LIN {X 0,Y 586.714,Z 168.831,A -85,B 0,C 180,E1 28018.701,E2 28018.701} C_VEL
LIN {X 0,Y 586.122,Z 408.457,A -85,B 0,C 180,E1 28015.501,E2 28015.501} C_VEL
LIN {X 0,Y 586.025,Z 431.656,A -85,B 0,C 180,E1 28015.125,E2 28015.125} C_VEL
LIN {X 0,Y 585.851,Z 452.374,A -85,B 0,C 180,E1 28014.603,E2 28014.603} C_VEL
LIN {X 0,Y 585.663,Z 472.135,A -85,B 0,C 180,E1 28013.921,E2 28013.921} C_VEL
LIN {X 0,Y 585.449,Z 491.199,A -85,B 0,C 180,E1 28013.077,E2 28013.077} C_VEL
LIN {X 0,Y 585.208,Z 509.397,A -85,B 0,C 180,E1 28012.079,E2 28012.079} C_VEL
LIN {X 0,Y 584.95,Z 527.579,A -85,B 0,C 180,E1 28010.883,E2 28010.883} C_VEL
LIN {X 0,Y 584.711,Z 544.758,A -85,B 0,C 180,E1 28009.536,E2 28009.536} C_VEL
LIN {X 0,Y 584.501,Z 560.932,A -85,B 0,C 180,E1 28008.037,E2 28008.037} C_VEL
LIN {X 0,Y 584.329,Z 575.047,A -85,B 0,C 180,E1 28006.502,E2 28006.502} C_VEL
LIN {X 0,Y 584.202,Z 587.854,A -85,B 0,C 180,E1 28004.876,E2 28004.876} C_VEL
LIN {X 0,Y 584.091,Z 599.923,A -85,B 0,C 180,E1 28003.06,E2 28003.06} C_VEL
LIN {X 0,Y 584.011,Z 610.394,A -85,B 0,C 180,E1 28001.155,E2 28001.155} C_VEL
LIN {X 0,Y 583.958,Z 618.872,A -85,B 0,C 180,E1 27999.262,E2 27999.262} C_VEL
LIN {X 0,Y 583.926,Z 625.897,A -85,B 0,C 180,E1 27997.28,E2 27997.28} C_VEL
LIN {X 0,Y 583.911,Z 631.143,A -85,B 0,C 180,E1 27995.306,E2 27995.306} C_VEL
LIN {X 0,Y 583.905,Z 634.713,A -85,B 0,C 180,E1 27993.336,E2 27993.336} C_VEL
LIN {X 0,Y 583.904,Z 636.639,A -85,B 0,C 180,E1 27991.276,E2 27991.276} C_VEL
LIN {X 0,Y 583.904,Z 636.852,A -85,B 0,C 180,E1 27989.314,E2 27989.314} C_VEL
LIN {X 0,Y 583.91,Z 635.393,A -85,B 0,C 180,E1 27987.253,E2 27987.253} C_VEL
LIN {X 0,Y 583.919,Z 632.17,A -85,B 0,C 180,E1 27985.188,E2 27985.188} C_VEL
LIN {X 0,Y 583.932,Z 627.416,A -85,B 0,C 180,E1 27983.215,E2 27983.215} C_VEL
LIN {X 0,Y 583.952,Z 620.853,A -85,B 0,C 180,E1 27981.235,E2 27981.235} C_VEL
LIN {X 0,Y 583.985,Z 612.797,A -85,B 0,C 180,E1 27979.345,E2 27979.345} C_VEL
LIN {X 0,Y 584.047,Z 602.84,A -85,B 0,C 180,E1 27977.443,E2 27977.443} C_VEL
LIN {X 0,Y 584.154,Z 591.394,A -85,B 0,C 180,E1 27975.63,E2 27975.63} C_VEL
LIN {X 0,Y 584.3,Z 578.453,A -85,B 0,C 180,E1 27973.907,E2 27973.907} C_VEL
LIN {X 0,Y 584.47,Z 563.98,A -85,B 0,C 180,E1 27972.272,E2 27972.272} C_VEL
LIN {X 0,Y 584.684,Z 548.453,A -85,B 0,C 180,E1 27970.781,E2 27970.781} C_VEL
LIN {X 0,Y 584.922,Z 531.283,A -85,B 0,C 180,E1 27969.383,E2 27969.383} C_VEL
LIN {X 0,Y 585.172,Z 512.918,A -85,B 0,C 180,E1 27968.132,E2 27968.132} C_VEL
LIN {X 0,Y 585.387,Z 494.302,A -85,B 0,C 180,E1 27967.082,E2 27967.082} C_VEL
LIN {X 0,Y 585.614,Z 475.711,A -85,B 0,C 180,E1 27966.227,E2 27966.227} C_VEL
LIN {X 0,Y 585.837,Z 455.081,A -85,B 0,C 180,E1 27965.48,E2 27965.48} C_VEL
LIN {X 0,Y 586.013,Z 435.161,A -85,B 0,C 180,E1 27964.947,E2 27964.947} C_VEL
LIN {X 0,Y 586.11,Z 414.501,A -85,B 0,C 180,E1 27964.579,E2 27964.579} C_VEL
LIN {X 0,Y 586.685,Z 176.57,A -85,B 0,C 180,E1 27961.403,E2 27961.403} C_VEL
LIN {X 0,Y 586.477,Z 165.201,A -85,B 0,C 180,E1 27961.237,E2 27961.237} C_VEL
LIN {X 0,Y 586.085,Z 162.496,A -85,B 0,C 180,E1 27961.161,E2 27961.161} C_VEL
LIN {X 0,Y 586.484,Z 115.163,A -85,B 0,C 180,E1 27958.212,E2 27958.212} C_VEL
LIN {X 0,Y 586.557,Z 103.347,A -85,B 0,C 180,E1 27957.46,E2 27957.46} C_VEL
LIN {X 0,Y 584.042,Z 96.734,A -85,B 0,C 180,E1 27956.871,E2 27956.871} C_VEL
LIN {X 0,Y 584.072,Z 96.733,A -85,B 0,C 180,E1 27953.68,E2 27953.68} C_VEL
LIN {X 0,Y 584.05,Z 96.728,A -85,B 0,C 180,E1 27950.696,E2 27950.696} C_VEL
LIN {X 0,Y 584.045,Z 96.731,A -85,B 0,C 180,E1 27947.403,E2 27947.403} C_VEL
LIN {X 0,Y 584.093,Z 96.728,A -85,B 0,C 180,E1 27944.3,E2 27944.3} C_VEL
LIN {X 0,Y 584.035,Z 96.729,A -85,B 0,C 180,E1 27941.127,E2 27941.127} C_VEL
LIN {X 0,Y 584.095,Z 96.723,A -85,B 0,C 180,E1 27938.043,E2 27938.043} C_VEL
LIN {X 0,Y 584.039,Z 96.729,A -85,B 0,C 180,E1 27934.913,E2 27934.913} C_VEL
LIN {X 0,Y 584.045,Z 96.731,A -85,B 0,C 180,E1 27931.591,E2 27931.591} C_VEL
LIN {X 0,Y 584.075,Z 96.727,A -85,B 0,C 180,E1 27928.529,E2 27928.529} C_VEL
LIN {X 0,Y 584.032,Z 96.729,A -85,B 0,C 180,E1 27925.322,E2 27925.322} C_VEL
LIN {X 0,Y 584.096,Z 96.731,A -85,B 0,C 180,E1 27922.17,E2 27922.17} C_VEL
LIN {X 0,Y 584.034,Z 96.727,A -85,B 0,C 180,E1 27919.086,E2 27919.086} C_VEL
LIN {X 0,Y 584.048,Z 96.731,A -85,B 0,C 180,E1 27915.795,E2 27915.795} C_VEL
LIN {X 0,Y 584.048,Z 96.726,A -85,B 0,C 180,E1 27912.859,E2 27912.859} C_VEL
LIN {X 0,Y 584.031,Z 96.73,A -85,B 0,C 180,E1 27909.567,E2 27909.567} C_VEL
LIN {X 0,Y 584.096,Z 96.726,A -85,B 0,C 180,E1 27906.487,E2 27906.487} C_VEL
LIN {X 0,Y 584.027,Z 96.73,A -85,B 0,C 180,E1 27903.337,E2 27903.337} C_VEL
LIN {X 0,Y 584.076,Z 96.731,A -85,B 0,C 180,E1 27900.196,E2 27900.196} C_VEL
LIN {X 0,Y 584.032,Z 96.73,A -85,B 0,C 180,E1 27897.154,E2 27897.154} C_VEL
LIN {X 0,Y 584.032,Z 96.73,A -85,B 0,C 180,E1 27893.808,E2 27893.808} C_VEL
LIN {X 0,Y 584.06,Z 96.73,A -85,B 0,C 180,E1 27890.839,E2 27890.839} C_VEL
LIN {X 0,Y 584.023,Z 96.729,A -85,B 0,C 180,E1 27887.643,E2 27887.643} C_VEL
LIN {X 0,Y 584.077,Z 96.728,A -85,B 0,C 180,E1 27886.731,E2 27886.731} C_VEL
LIN {X 0,Y 583.129,Z 96.853,A -85,B 0,C 180,E1 27885.975,E2 27885.975} C_VEL
LIN {X 0,Y 576.616,Z 97.654,A -85,B 0,C 180,E1 27883.855,E2 27883.855} C_VEL
LIN {X 0,Y 576.087,Z 97.718,A -85,B 0,C 180,E1 27883.302,E2 27883.302} C_VEL
LIN {X 0,Y 576.097,Z 97.721,A -85,B 0,C 180,E1 27880.007,E2 27880.007} C_VEL
LIN {X 0,Y 576.11,Z 97.718,A -85,B 0,C 180,E1 27877.014,E2 27877.014} C_VEL
LIN {X 0,Y 576.084,Z 97.72,A -85,B 0,C 180,E1 27873.805,E2 27873.805} C_VEL
LIN {X 0,Y 576.149,Z 97.717,A -85,B 0,C 180,E1 27870.699,E2 27870.699} C_VEL
LIN {X 0,Y 576.078,Z 97.719,A -85,B 0,C 180,E1 27867.567,E2 27867.567} C_VEL
LIN {X 0,Y 576.128,Z 97.72,A -85,B 0,C 180,E1 27864.452,E2 27864.452} C_VEL
LIN {X 0,Y 576.089,Z 97.72,A -85,B 0,C 180,E1 27861.331,E2 27861.331} C_VEL
LIN {X 0,Y 576.086,Z 97.721,A -85,B 0,C 180,E1 27858.071,E2 27858.071} C_VEL
LIN {X 0,Y 576.115,Z 97.719,A -85,B 0,C 180,E1 27855.06,E2 27855.06} C_VEL
LIN {X 0,Y 576.077,Z 97.722,A -85,B 0,C 180,E1 27851.876,E2 27851.876} C_VEL
LIN {X 0,Y 576.157,Z 97.721,A -85,B 0,C 180,E1 27848.79,E2 27848.79} C_VEL
LIN {X 0,Y 576.08,Z 97.721,A -85,B 0,C 180,E1 27845.673,E2 27845.673} C_VEL
LIN {X 0,Y 576.109,Z 97.724,A -85,B 0,C 180,E1 27842.43,E2 27842.43} C_VEL
LIN {X 0,Y 576.088,Z 97.795,A -85,B 0,C 180,E1 27839.824,E2 27839.824} C_VEL
LIN {X 0,Y 578.546,Z 105.77,A -85,B 0,C 180,E1 27839.016,E2 27839.016} C_VEL
LIN {X 0,Y 577.999,Z 143.994,A -85,B 0,C 180,E1 27835.953,E2 27835.953} C_VEL
LIN {X 0,Y 577.653,Z 175.774,A -85,B 0,C 180,E1 27833.508,E2 27833.508} C_VEL
LIN {X 0,Y 578.35,Z 181.85,A -85,B 0,C 180,E1 27833.398,E2 27833.398} C_VEL
LIN {X 0,Y 577.837,Z 384.429,A -85,B 0,C 180,E1 27830.729,E2 27830.729} C_VEL
LIN {X 0,Y 577.687,Z 403.356,A -85,B 0,C 180,E1 27830.29,E2 27830.29} C_VEL
LIN {X 0,Y 577.5,Z 421.605,A -85,B 0,C 180,E1 27829.678,E2 27829.678} C_VEL
LIN {X 0,Y 577.269,Z 439.198,A -85,B 0,C 180,E1 27828.898,E2 27828.898} C_VEL
LIN {X 0,Y 577.04,Z 455.969,A -85,B 0,C 180,E1 27827.959,E2 27827.959} C_VEL
LIN {X 0,Y 576.809,Z 471.559,A -85,B 0,C 180,E1 27826.891,E2 27826.891} C_VEL
LIN {X 0,Y 576.58,Z 486.636,A -85,B 0,C 180,E1 27825.643,E2 27825.643} C_VEL
LIN {X 0,Y 576.378,Z 500.546,A -85,B 0,C 180,E1 27824.26,E2 27824.26} C_VEL
LIN {X 0,Y 576.212,Z 513.352,A -85,B 0,C 180,E1 27822.73,E2 27822.73} C_VEL
LIN {X 0,Y 576.088,Z 524.59,A -85,B 0,C 180,E1 27821.107,E2 27821.107} C_VEL
LIN {X 0,Y 576.002,Z 534.283,A -85,B 0,C 180,E1 27819.39,E2 27819.39} C_VEL
LIN {X 0,Y 575.957,Z 542,A -85,B 0,C 180,E1 27817.681,E2 27817.681} C_VEL
LIN {X 0,Y 575.927,Z 548.347,A -85,B 0,C 180,E1 27815.856,E2 27815.856} C_VEL
LIN {X 0,Y 575.92,Z 552.989,A -85,B 0,C 180,E1 27813.981,E2 27813.981} C_VEL
LIN {X 0,Y 575.917,Z 555.852,A -85,B 0,C 180,E1 27812.089,E2 27812.089} C_VEL
LIN {X 0,Y 575.911,Z 556.952,A -85,B 0,C 180,E1 27810.198,E2 27810.198} C_VEL
LIN {X 0,Y 575.914,Z 556.311,A -85,B 0,C 180,E1 27808.308,E2 27808.308} C_VEL
LIN {X 0,Y 575.909,Z 553.916,A -85,B 0,C 180,E1 27806.416,E2 27806.416} C_VEL
LIN {X 0,Y 575.922,Z 549.956,A -85,B 0,C 180,E1 27804.62,E2 27804.62} C_VEL
LIN {X 0,Y 575.939,Z 544.27,A -85,B 0,C 180,E1 27802.819,E2 27802.819} C_VEL
LIN {X 0,Y 575.981,Z 537.168,A -85,B 0,C 180,E1 27801.112,E2 27801.112} C_VEL
LIN {X 0,Y 576.056,Z 528.191,A -85,B 0,C 180,E1 27799.398,E2 27799.398} C_VEL
LIN {X 0,Y 576.167,Z 517.752,A -85,B 0,C 180,E1 27797.777,E2 27797.777} C_VEL
LIN {X 0,Y 576.31,Z 505.869,A -85,B 0,C 180,E1 27796.249,E2 27796.249} C_VEL
LIN {X 0,Y 576.498,Z 492.507,A -85,B 0,C 180,E1 27794.817,E2 27794.817} C_VEL
LIN {X 0,Y 576.723,Z 477.51,A -85,B 0,C 180,E1 27793.481,E2 27793.481} C_VEL
LIN {X 0,Y 576.961,Z 461.313,A -85,B 0,C 180,E1 27792.293,E2 27792.293} C_VEL
LIN {X 0,Y 577.198,Z 444.899,A -85,B 0,C 180,E1 27791.308,E2 27791.308} C_VEL
LIN {X 0,Y 577.43,Z 427.61,A -85,B 0,C 180,E1 27790.476,E2 27790.476} C_VEL
LIN {X 0,Y 577.635,Z 409.432,A -85,B 0,C 180,E1 27789.803,E2 27789.803} C_VEL
LIN {X 0,Y 577.794,Z 390.88,A -85,B 0,C 180,E1 27789.311,E2 27789.311} C_VEL
LIN {X 0,Y 577.893,Z 370.714,A -85,B 0,C 180,E1 27788.977,E2 27788.977} C_VEL
LIN {X 0,Y 578.232,Z 179.106,A -85,B 0,C 180,E1 27786.471,E2 27786.471} C_VEL
LIN {X 0,Y 577.601,Z 175.101,A -85,B 0,C 180,E1 27786.375,E2 27786.375} C_VEL
LIN {X 0,Y 578.093,Z 134.758,A -85,B 0,C 180,E1 27783.22,E2 27783.22} C_VEL
LIN {X 0,Y 578.526,Z 105.079,A -85,B 0,C 180,E1 27780.831,E2 27780.831} C_VEL
LIN {X 0,Y 576.084,Z 97.726,A -85,B 0,C 180,E1 27780.066,E2 27780.066} C_VEL
LIN {X 0,Y 576.121,Z 97.719,A -85,B 0,C 180,E1 27776.86,E2 27776.86} C_VEL
LIN {X 0,Y 576.135,Z 97.721,A -85,B 0,C 180,E1 27773.715,E2 27773.715} C_VEL
LIN {X 0,Y 576.115,Z 97.71,A -85,B 0,C 180,E1 27770.562,E2 27770.562} C_VEL
LIN {X 0,Y 576.158,Z 97.714,A -85,B 0,C 180,E1 27767.376,E2 27767.376} C_VEL
LIN {X 0,Y 576.155,Z 97.72,A -85,B 0,C 180,E1 27764.072,E2 27764.072} C_VEL
LIN {X 0,Y 576.14,Z 97.716,A -85,B 0,C 180,E1 27760.733,E2 27760.733} C_VEL
LIN {X 0,Y 576.149,Z 97.713,A -85,B 0,C 180,E1 27757.525,E2 27757.525} C_VEL
LIN {X 0,Y 576.142,Z 97.72,A -85,B 0,C 180,E1 27754.214,E2 27754.214} C_VEL
LIN {X 0,Y 576.158,Z 97.72,A -85,B 0,C 180,E1 27750.909,E2 27750.909} C_VEL
LIN {X 0,Y 576.141,Z 97.757,A -85,B 0,C 180,E1 27749.631,E2 27749.631} C_VEL
LIN {X 0,Y 578.217,Z 105.123,A -85,B 0,C 180,E1 27748.957,E2 27748.957} C_VEL
LIN {X 0,Y 577.914,Z 144.603,A -85,B 0,C 180,E1 27745.886,E2 27745.886} C_VEL
LIN {X 0,Y 577.621,Z 175.862,A -85,B 0,C 180,E1 27743.509,E2 27743.509} C_VEL
LIN {X 0,Y 578.323,Z 181.943,A -85,B 0,C 180,E1 27743.398,E2 27743.398} C_VEL
LIN {X 0,Y 577.84,Z 384.232,A -85,B 0,C 180,E1 27740.732,E2 27740.732} C_VEL
LIN {X 0,Y 577.685,Z 402.976,A -85,B 0,C 180,E1 27740.297,E2 27740.297} C_VEL
LIN {X 0,Y 577.519,Z 420.285,A -85,B 0,C 180,E1 27739.731,E2 27739.731} C_VEL
LIN {X 0,Y 577.286,Z 437.662,A -85,B 0,C 180,E1 27738.972,E2 27738.972} C_VEL
LIN {X 0,Y 577.052,Z 455.018,A -85,B 0,C 180,E1 27738.017,E2 27738.017} C_VEL
LIN {X 0,Y 576.823,Z 471.07,A -85,B 0,C 180,E1 27736.931,E2 27736.931} C_VEL
LIN {X 0,Y 576.585,Z 486.027,A -85,B 0,C 180,E1 27735.695,E2 27735.695} C_VEL
LIN {X 0,Y 576.401,Z 499.639,A -85,B 0,C 180,E1 27734.363,E2 27734.363} C_VEL
LIN {X 0,Y 576.222,Z 512.539,A -85,B 0,C 180,E1 27732.833,E2 27732.833} C_VEL
LIN {X 0,Y 576.102,Z 523.356,A -85,B 0,C 180,E1 27731.306,E2 27731.306} C_VEL
LIN {X 0,Y 576.014,Z 533.232,A -85,B 0,C 180,E1 27729.593,E2 27729.593} C_VEL
LIN {X 0,Y 575.954,Z 541.206,A -85,B 0,C 180,E1 27727.883,E2 27727.883} C_VEL
LIN {X 0,Y 575.927,Z 547.971,A -85,B 0,C 180,E1 27725.979,E2 27725.979} C_VEL
LIN {X 0,Y 575.914,Z 552.591,A -85,B 0,C 180,E1 27724.182,E2 27724.182} C_VEL
LIN {X 0,Y 575.913,Z 555.743,A -85,B 0,C 180,E1 27722.189,E2 27722.189} C_VEL
LIN {X 0,Y 575.913,Z 556.936,A -85,B 0,C 180,E1 27720.299,E2 27720.299} C_VEL
LIN {X 0,Y 575.91,Z 556.313,A -85,B 0,C 180,E1 27718.309,E2 27718.309} C_VEL
LIN {X 0,Y 575.918,Z 554.069,A -85,B 0,C 180,E1 27716.517,E2 27716.517} C_VEL
LIN {X 0,Y 575.922,Z 549.975,A -85,B 0,C 180,E1 27714.621,E2 27714.621} C_VEL
LIN {X 0,Y 575.942,Z 544.257,A -85,B 0,C 180,E1 27712.82,E2 27712.82} C_VEL
LIN {X 0,Y 575.988,Z 536.728,A -85,B 0,C 180,E1 27711.012,E2 27711.012} C_VEL
LIN {X 0,Y 576.058,Z 528.17,A -85,B 0,C 180,E1 27709.398,E2 27709.398} C_VEL
LIN {X 0,Y 576.178,Z 517.139,A -85,B 0,C 180,E1 27707.687,E2 27707.687} C_VEL
LIN {X 0,Y 576.321,Z 504.976,A -85,B 0,C 180,E1 27706.148,E2 27706.148} C_VEL
LIN {X 0,Y 576.511,Z 491.443,A -85,B 0,C 180,E1 27704.715,E2 27704.715} C_VEL
LIN {X 0,Y 576.709,Z 477.443,A -85,B 0,C 180,E1 27703.481,E2 27703.481} C_VEL
LIN {X 0,Y 576.952,Z 462.1,A -85,B 0,C 180,E1 27702.346,E2 27702.346} C_VEL
LIN {X 0,Y 577.177,Z 445.959,A -85,B 0,C 180,E1 27701.368,E2 27701.368} C_VEL
LIN {X 0,Y 577.41,Z 428.793,A -85,B 0,C 180,E1 27700.529,E2 27700.529} C_VEL
LIN {X 0,Y 577.605,Z 411.69,A -85,B 0,C 180,E1 27699.877,E2 27699.877} C_VEL
LIN {X 0,Y 577.766,Z 392.811,A -85,B 0,C 180,E1 27699.355,E2 27699.355} C_VEL
LIN {X 0,Y 577.89,Z 373.954,A -85,B 0,C 180,E1 27699.019,E2 27699.019} C_VEL
LIN {X 0,Y 578.245,Z 179.115,A -85,B 0,C 180,E1 27696.472,E2 27696.472} C_VEL
LIN {X 0,Y 577.585,Z 175.11,A -85,B 0,C 180,E1 27696.375,E2 27696.375} C_VEL
LIN {X 0,Y 577.951,Z 136.16,A -85,B 0,C 180,E1 27693.38,E2 27693.38} C_VEL
LIN {X 0,Y 578.003,Z 114.036,A -85,B 0,C 180,E1 27691.703,E2 27691.703} C_VEL
LIN {X 0,Y 577.718,Z 103.475,A -85,B 0,C 180,E1 27690.928,E2 27690.928} C_VEL
LIN {X 0,Y 576.121,Z 97.721,A -85,B 0,C 180,E1 27690.441,E2 27690.441} C_VEL
LIN {X 0,Y 576.162,Z 97.72,A -85,B 0,C 180,E1 27687.219,E2 27687.219} C_VEL
LIN {X 0,Y 576.133,Z 97.717,A -85,B 0,C 180,E1 27683.962,E2 27683.962} C_VEL
LIN {X 0,Y 576.101,Z 97.72,A -85,B 0,C 180,E1 27680.693,E2 27680.693} C_VEL
LIN {X 0,Y 576.153,Z 97.721,A -85,B 0,C 180,E1 27677.523,E2 27677.523} C_VEL
LIN {X 0,Y 576.094,Z 97.721,A -85,B 0,C 180,E1 27674.383,E2 27674.383} C_VEL
LIN {X 0,Y 576.084,Z 97.722,A -85,B 0,C 180,E1 27671.001,E2 27671.001} C_VEL
LIN {X 0,Y 576.153,Z 97.721,A -85,B 0,C 180,E1 27667.904,E2 27667.904} C_VEL
LIN {X 0,Y 576.096,Z 97.723,A -85,B 0,C 180,E1 27664.7,E2 27664.7} C_VEL
LIN {X 0,Y 576.135,Z 97.75,A -85,B 0,C 180,E1 27663.573,E2 27663.573} C_VEL
LIN {X 0,Y 579.556,Z 106.935,A -85,B 0,C 180,E1 27662.748,E2 27662.748} C_VEL
LIN {X 0,Y 578.949,Z 154.809,A -85,B 0,C 180,E1 27659.714,E2 27659.714} C_VEL
LIN {X 0,Y 578.961,Z 163.557,A -85,B 0,C 180,E1 27659.195,E2 27659.195} C_VEL
LIN {X 0,Y 579.691,Z 169.722,A -85,B 0,C 180,E1 27659.069,E2 27659.069} C_VEL
LIN {X 0,Y 578.899,Z 409.209,A -85,B 0,C 180,E1 27655.832,E2 27655.832} C_VEL
LIN {X 0,Y 578.766,Z 431.846,A -85,B 0,C 180,E1 27655.459,E2 27655.459} C_VEL
LIN {X 0,Y 578.532,Z 452.639,A -85,B 0,C 180,E1 27654.927,E2 27654.927} C_VEL
LIN {X 0,Y 578.29,Z 472.133,A -85,B 0,C 180,E1 27654.245,E2 27654.245} C_VEL
LIN {X 0,Y 577.996,Z 491.203,A -85,B 0,C 180,E1 27653.392,E2 27653.392} C_VEL
LIN {X 0,Y 577.66,Z 510.29,A -85,B 0,C 180,E1 27652.33,E2 27652.33} C_VEL
LIN {X 0,Y 577.326,Z 527.635,A -85,B 0,C 180,E1 27651.168,E2 27651.168} C_VEL
LIN {X 0,Y 577.008,Z 544.936,A -85,B 0,C 180,E1 27649.792,E2 27649.792} C_VEL
LIN {X 0,Y 576.715,Z 561.438,A -85,B 0,C 180,E1 27648.237,E2 27648.237} C_VEL
LIN {X 0,Y 576.472,Z 575.897,A -85,B 0,C 180,E1 27646.63,E2 27646.63} C_VEL
LIN {X 0,Y 576.284,Z 589.161,A -85,B 0,C 180,E1 27644.895,E2 27644.895} C_VEL
LIN {X 0,Y 576.149,Z 600.524,A -85,B 0,C 180,E1 27643.141,E2 27643.141} C_VEL
LIN {X 0,Y 576.043,Z 610.908,A -85,B 0,C 180,E1 27641.21,E2 27641.21} C_VEL
LIN {X 0,Y 575.973,Z 619.278,A -85,B 0,C 180,E1 27639.291,E2 27639.291} C_VEL
LIN {X 0,Y 575.932,Z 625.897,A -85,B 0,C 180,E1 27637.382,E2 27637.382} C_VEL
LIN {X 0,Y 575.912,Z 631.143,A -85,B 0,C 180,E1 27635.38,E2 27635.38} C_VEL
LIN {X 0,Y 575.906,Z 634.745,A -85,B 0,C 180,E1 27633.357,E2 27633.357} C_VEL
LIN {X 0,Y 575.903,Z 636.639,A -85,B 0,C 180,E1 27631.294,E2 27631.294} C_VEL
LIN {X 0,Y 575.904,Z 636.852,A -85,B 0,C 180,E1 27629.304,E2 27629.304} C_VEL
LIN {X 0,Y 575.912,Z 635.393,A -85,B 0,C 180,E1 27627.214,E2 27627.214} C_VEL
LIN {X 0,Y 575.921,Z 632.17,A -85,B 0,C 180,E1 27625.121,E2 27625.121} C_VEL
LIN {X 0,Y 575.938,Z 627.416,A -85,B 0,C 180,E1 27623.121,E2 27623.121} C_VEL
LIN {X 0,Y 575.967,Z 620.853,A -85,B 0,C 180,E1 27621.113,E2 27621.113} C_VEL
LIN {X 0,Y 576.017,Z 612.797,A -85,B 0,C 180,E1 27619.196,E2 27619.196} C_VEL
LIN {X 0,Y 576.102,Z 602.842,A -85,B 0,C 180,E1 27617.267,E2 27617.267} C_VEL
LIN {X 0,Y 576.247,Z 591.395,A -85,B 0,C 180,E1 27615.429,E2 27615.429} C_VEL
LIN {X 0,Y 576.439,Z 578.452,A -85,B 0,C 180,E1 27613.681,E2 27613.681} C_VEL
LIN {X 0,Y 576.673,Z 563.98,A -85,B 0,C 180,E1 27612.024,E2 27612.024} C_VEL
LIN {X 0,Y 576.961,Z 548.486,A -85,B 0,C 180,E1 27610.516,E2 27610.516} C_VEL
LIN {X 0,Y 577.284,Z 531.284,A -85,B 0,C 180,E1 27609.097,E2 27609.097} C_VEL
LIN {X 0,Y 577.624,Z 512.914,A -85,B 0,C 180,E1 27607.831,E2 27607.831} C_VEL
LIN {X 0,Y 577.925,Z 494.298,A -85,B 0,C 180,E1 27606.769,E2 27606.769} C_VEL
LIN {X 0,Y 578.224,Z 475.18,A -85,B 0,C 180,E1 27605.881,E2 27605.881} C_VEL
LIN {X 0,Y 578.517,Z 454.709,A -85,B 0,C 180,E1 27605.137,E2 27605.137} C_VEL
LIN {X 0,Y 578.752,Z 434.609,A -85,B 0,C 180,E1 27604.599,E2 27604.599} C_VEL
LIN {X 0,Y 578.886,Z 413.866,A -85,B 0,C 180,E1 27604.23,E2 27604.23} C_VEL
LIN {X 0,Y 579.665,Z 175.552,A -85,B 0,C 180,E1 27601.01,E2 27601.01} C_VEL
LIN {X 0,Y 579.444,Z 166.395,A -85,B 0,C 180,E1 27600.871,E2 27600.871} C_VEL
LIN {X 0,Y 578.855,Z 162.496,A -85,B 0,C 180,E1 27600.766,E2 27600.766} C_VEL
LIN {X 0,Y 579.405,Z 116.064,A -85,B 0,C 180,E1 27597.835,E2 27597.835} C_VEL
LIN {X 0,Y 579.556,Z 106.958,A -85,B 0,C 180,E1 27597.253,E2 27597.253} C_VEL
LIN {X 0,Y 576.134,Z 97.72,A -85,B 0,C 180,E1 27596.41,E2 27596.41} C_VEL
LIN {X 0,Y 576.102,Z 97.721,A -85,B 0,C 180,E1 27593.219,E2 27593.219} C_VEL
LIN {X 0,Y 576.164,Z 97.718,A -85,B 0,C 180,E1 27590.053,E2 27590.053} C_VEL
LIN {X 0,Y 576.103,Z 97.719,A -85,B 0,C 180,E1 27586.859,E2 27586.859} C_VEL
LIN {X 0,Y 576.108,Z 97.718,A -85,B 0,C 180,E1 27583.495,E2 27583.495} C_VEL
LIN {X 0,Y 576.152,Z 97.716,A -85,B 0,C 180,E1 27580.339,E2 27580.339} C_VEL
LIN {X 0,Y 576.095,Z 97.715,A -85,B 0,C 180,E1 27577.155,E2 27577.155} C_VEL
LIN {X 0,Y 576.143,Z 97.718,A -85,B 0,C 180,E1 27573.95,E2 27573.95} C_VEL
LIN {X 0,Y 576.102,Z 97.718,A -85,B 0,C 180,E1 27570.912,E2 27570.912} C_VEL
LIN {X 0,Y 576.101,Z 97.719,A -85,B 0,C 180,E1 27567.519,E2 27567.519} C_VEL
LIN {X 0,Y 576.151,Z 97.717,A -85,B 0,C 180,E1 27564.395,E2 27564.395} C_VEL
LIN {X 0,Y 576.092,Z 97.719,A -85,B 0,C 180,E1 27561.252,E2 27561.252} C_VEL
LIN {X 0,Y 576.144,Z 97.72,A -85,B 0,C 180,E1 27558.098,E2 27558.098} C_VEL
LIN {X 0,Y 576.1,Z 97.718,A -85,B 0,C 180,E1 27554.987,E2 27554.987} C_VEL
LIN {X 0,Y 576.095,Z 97.719,A -85,B 0,C 180,E1 27551.614,E2 27551.614} C_VEL
LIN {X 0,Y 576.152,Z 97.718,A -85,B 0,C 180,E1 27548.482,E2 27548.482} C_VEL
LIN {X 0,Y 576.088,Z 97.719,A -85,B 0,C 180,E1 27545.378,E2 27545.378} C_VEL
LIN {X 0,Y 576.137,Z 97.717,A -85,B 0,C 180,E1 27542.188,E2 27542.188} C_VEL
LIN {X 0,Y 576.095,Z 97.718,A -85,B 0,C 180,E1 27539.105,E2 27539.105} C_VEL
LIN {X 0,Y 576.095,Z 97.718,A -85,B 0,C 180,E1 27535.82,E2 27535.82} C_VEL
LIN {X 0,Y 576.122,Z 97.717,A -85,B 0,C 180,E1 27532.822,E2 27532.822} C_VEL
LIN {X 0,Y 576.084,Z 97.718,A -85,B 0,C 180,E1 27529.601,E2 27529.601} C_VEL
LIN {X 0,Y 576.154,Z 97.72,A -85,B 0,C 180,E1 27526.451,E2 27526.451} C_VEL
LIN {X 0,Y 576.087,Z 97.718,A -85,B 0,C 180,E1 27523.302,E2 27523.302} C_VEL
LIN {X 0,Y 575.122,Z 97.845,A -85,B 0,C 180,E1 27522.536,E2 27522.536} C_VEL
LIN {X 0,Y 568.601,Z 98.659,A -85,B 0,C 180,E1 27520.33,E2 27520.33} C_VEL
LIN {X 0,Y 568.148,Z 98.709,A -85,B 0,C 180,E1 27519.825,E2 27519.825} C_VEL
LIN {X 0,Y 568.211,Z 98.705,A -85,B 0,C 180,E1 27516.676,E2 27516.676} C_VEL
LIN {X 0,Y 568.142,Z 98.709,A -85,B 0,C 180,E1 27513.561,E2 27513.561} C_VEL
LIN {X 0,Y 568.185,Z 98.71,A -85,B 0,C 180,E1 27510.364,E2 27510.364} C_VEL
LIN {X 0,Y 568.153,Z 98.708,A -85,B 0,C 180,E1 27507.266,E2 27507.266} C_VEL
LIN {X 0,Y 568.146,Z 98.709,A -85,B 0,C 180,E1 27503.999,E2 27503.999} C_VEL
LIN {X 0,Y 568.204,Z 98.709,A -85,B 0,C 180,E1 27500.822,E2 27500.822} C_VEL
LIN {X 0,Y 568.137,Z 98.71,A -85,B 0,C 180,E1 27497.658,E2 27497.658} C_VEL
LIN {X 0,Y 568.179,Z 98.711,A -85,B 0,C 180,E1 27494.457,E2 27494.457} C_VEL
LIN {X 0,Y 568.148,Z 98.711,A -85,B 0,C 180,E1 27491.429,E2 27491.429} C_VEL
LIN {X 0,Y 568.147,Z 98.709,A -85,B 0,C 180,E1 27488.125,E2 27488.125} C_VEL
LIN {X 0,Y 568.196,Z 98.709,A -85,B 0,C 180,E1 27485.005,E2 27485.005} C_VEL
LIN {X 0,Y 568.14,Z 98.714,A -85,B 0,C 180,E1 27481.867,E2 27481.867} C_VEL
LIN {X 0,Y 568.181,Z 98.929,A -85,B 0,C 180,E1 27480.226,E2 27480.226} C_VEL
LIN {X 0,Y 571.286,Z 108.519,A -85,B 0,C 180,E1 27479.228,E2 27479.228} C_VEL
LIN {X 0,Y 570.598,Z 147.207,A -85,B 0,C 180,E1 27476.092,E2 27476.092} C_VEL
LIN {X 0,Y 570.154,Z 175.718,A -85,B 0,C 180,E1 27473.852,E2 27473.852} C_VEL
LIN {X 0,Y 571.026,Z 182.769,A -85,B 0,C 180,E1 27473.71,E2 27473.71} C_VEL
LIN {X 0,Y 570.356,Z 384.462,A -85,B 0,C 180,E1 27471.014,E2 27471.014} C_VEL
LIN {X 0,Y 570.165,Z 403.441,A -85,B 0,C 180,E1 27470.568,E2 27470.568} C_VEL
LIN {X 0,Y 569.93,Z 421.618,A -85,B 0,C 180,E1 27469.951,E2 27469.951} C_VEL
LIN {X 0,Y 569.64,Z 439.206,A -85,B 0,C 180,E1 27469.161,E2 27469.161} C_VEL
LIN {X 0,Y 569.347,Z 455.902,A -85,B 0,C 180,E1 27468.215,E2 27468.215} C_VEL
LIN {X 0,Y 569.044,Z 472.093,A -85,B 0,C 180,E1 27467.087,E2 27467.087} C_VEL
LIN {X 0,Y 568.754,Z 487.196,A -85,B 0,C 180,E1 27465.812,E2 27465.812} C_VEL
LIN {X 0,Y 568.515,Z 500.551,A -85,B 0,C 180,E1 27464.461,E2 27464.461} C_VEL
LIN {X 0,Y 568.302,Z 513.357,A -85,B 0,C 180,E1 27462.91,E2 27462.91} C_VEL
LIN {X 0,Y 568.138,Z 524.593,A -85,B 0,C 180,E1 27461.264,E2 27461.264} C_VEL
LIN {X 0,Y 568.028,Z 534.286,A -85,B 0,C 180,E1 27459.523,E2 27459.523} C_VEL
LIN {X 0,Y 567.968,Z 542.002,A -85,B 0,C 180,E1 27457.79,E2 27457.79} C_VEL
LIN {X 0,Y 567.933,Z 548.282,A -85,B 0,C 180,E1 27455.961,E2 27455.961} C_VEL
LIN {X 0,Y 567.919,Z 552.787,A -85,B 0,C 180,E1 27454.139,E2 27454.139} C_VEL
LIN {X 0,Y 567.915,Z 555.743,A -85,B 0,C 180,E1 27452.219,E2 27452.219} C_VEL
LIN {X 0,Y 567.909,Z 556.93,A -85,B 0,C 180,E1 27450.302,E2 27450.302} C_VEL
LIN {X 0,Y 567.914,Z 556.378,A -85,B 0,C 180,E1 27448.385,E2 27448.385} C_VEL
LIN {X 0,Y 567.908,Z 554.074,A -85,B 0,C 180,E1 27446.467,E2 27446.467} C_VEL
LIN {X 0,Y 567.924,Z 550.208,A -85,B 0,C 180,E1 27444.645,E2 27444.645} C_VEL
LIN {X 0,Y 567.945,Z 544.62,A -85,B 0,C 180,E1 27442.819,E2 27442.819} C_VEL
LIN {X 0,Y 567.998,Z 537.626,A -85,B 0,C 180,E1 27441.088,E2 27441.088} C_VEL
LIN {X 0,Y 568.091,Z 528.765,A -85,B 0,C 180,E1 27439.35,E2 27439.35} C_VEL
LIN {X 0,Y 568.229,Z 518.454,A -85,B 0,C 180,E1 27437.706,E2 27437.706} C_VEL
LIN {X 0,Y 568.406,Z 506.713,A -85,B 0,C 180,E1 27436.158,E2 27436.158} C_VEL
LIN {X 0,Y 568.639,Z 493.513,A -85,B 0,C 180,E1 27434.707,E2 27434.707} C_VEL
LIN {X 0,Y 568.92,Z 478.736,A -85,B 0,C 180,E1 27433.353,E2 27433.353} C_VEL
LIN {X 0,Y 569.224,Z 462.866,A -85,B 0,C 180,E1 27432.15,E2 27432.15} C_VEL
LIN {X 0,Y 569.536,Z 445.883,A -85,B 0,C 180,E1 27431.1,E2 27431.1} C_VEL
LIN {X 0,Y 569.826,Z 428.863,A -85,B 0,C 180,E1 27430.258,E2 27430.258} C_VEL
LIN {X 0,Y 570.091,Z 410.245,A -85,B 0,C 180,E1 27429.55,E2 27429.55} C_VEL
LIN {X 0,Y 570.295,Z 391.496,A -85,B 0,C 180,E1 27429.04,E2 27429.04} C_VEL
LIN {X 0,Y 570.421,Z 371.554,A -85,B 0,C 180,E1 27428.7,E2 27428.7} C_VEL
LIN {X 0,Y 570.928,Z 180.337,A -85,B 0,C 180,E1 27426.161,E2 27426.161} C_VEL
LIN {X 0,Y 570.09,Z 175.035,A -85,B 0,C 180,E1 27426.031,E2 27426.031} C_VEL
LIN {X 0,Y 570.769,Z 135.339,A -85,B 0,C 180,E1 27422.861,E2 27422.861} C_VEL
LIN {X 0,Y 571.288,Z 108.097,A -85,B 0,C 180,E1 27420.645,E2 27420.645} C_VEL
LIN {X 0,Y 568.169,Z 98.715,A -85,B 0,C 180,E1 27419.635,E2 27419.635} C_VEL
LIN {X 0,Y 568.156,Z 98.709,A -85,B 0,C 180,E1 27416.455,E2 27416.455} C_VEL
LIN {X 0,Y 568.222,Z 98.708,A -85,B 0,C 180,E1 27413.253,E2 27413.253} C_VEL
LIN {X 0,Y 568.197,Z 98.701,A -85,B 0,C 180,E1 27409.949,E2 27409.949} C_VEL
LIN {X 0,Y 568.186,Z 98.704,A -85,B 0,C 180,E1 27406.617,E2 27406.617} C_VEL
LIN {X 0,Y 568.218,Z 98.7,A -85,B 0,C 180,E1 27403.335,E2 27403.335} C_VEL
LIN {X 0,Y 568.213,Z 98.707,A -85,B 0,C 180,E1 27399.962,E2 27399.962} C_VEL
LIN {X 0,Y 568.214,Z 98.707,A -85,B 0,C 180,E1 27396.622,E2 27396.622} C_VEL
LIN {X 0,Y 568.218,Z 98.703,A -85,B 0,C 180,E1 27393.297,E2 27393.297} C_VEL
LIN {X 0,Y 568.185,Z 98.71,A -85,B 0,C 180,E1 27389.985,E2 27389.985} C_VEL
LIN {X 0,Y 570.781,Z 107.539,A -85,B 0,C 180,E1 27389.143,E2 27389.143} C_VEL
LIN {X 0,Y 570.435,Z 146.471,A -85,B 0,C 180,E1 27386.101,E2 27386.101} C_VEL
LIN {X 0,Y 570.08,Z 175.861,A -85,B 0,C 180,E1 27383.837,E2 27383.837} C_VEL
LIN {X 0,Y 570.98,Z 182.871,A -85,B 0,C 180,E1 27383.705,E2 27383.705} C_VEL
LIN {X 0,Y 570.356,Z 384.027,A -85,B 0,C 180,E1 27381.02,E2 27381.02} C_VEL
LIN {X 0,Y 570.167,Z 402.675,A -85,B 0,C 180,E1 27380.586,E2 27380.586} C_VEL
LIN {X 0,Y 569.952,Z 420.3,A -85,B 0,C 180,E1 27380.004,E2 27380.004} C_VEL
LIN {X 0,Y 569.666,Z 437.016,A -85,B 0,C 180,E1 27379.267,E2 27379.267} C_VEL
LIN {X 0,Y 569.378,Z 454.19,A -85,B 0,C 180,E1 27378.321,E2 27378.321} C_VEL
LIN {X 0,Y 569.086,Z 469.632,A -85,B 0,C 180,E1 27377.273,E2 27377.273} C_VEL
LIN {X 0,Y 568.789,Z 484.888,A -85,B 0,C 180,E1 27376.021,E2 27376.021} C_VEL
LIN {X 0,Y 568.547,Z 498.312,A -85,B 0,C 180,E1 27374.705,E2 27374.705} C_VEL
LIN {X 0,Y 568.336,Z 510.984,A -85,B 0,C 180,E1 27373.221,E2 27373.221} C_VEL
LIN {X 0,Y 568.178,Z 521.984,A -85,B 0,C 180,E1 27371.676,E2 27371.676} C_VEL
LIN {X 0,Y 568.054,Z 532.2,A -85,B 0,C 180,E1 27369.933,E2 27369.933} C_VEL
LIN {X 0,Y 567.985,Z 539.918,A -85,B 0,C 180,E1 27368.3,E2 27368.3} C_VEL
LIN {X 0,Y 567.946,Z 546.764,A -85,B 0,C 180,E1 27366.47,E2 27366.47} C_VEL
LIN {X 0,Y 567.919,Z 551.704,A -85,B 0,C 180,E1 27364.645,E2 27364.645} C_VEL
LIN {X 0,Y 567.915,Z 555.026,A -85,B 0,C 180,E1 27362.826,E2 27362.826} C_VEL
LIN {X 0,Y 567.909,Z 556.748,A -85,B 0,C 180,E1 27360.908,E2 27360.908} C_VEL
LIN {X 0,Y 567.912,Z 556.788,A -85,B 0,C 180,E1 27359.092,E2 27359.092} C_VEL
LIN {X 0,Y 567.909,Z 555.143,A -85,B 0,C 180,E1 27357.175,E2 27357.175} C_VEL
LIN {X 0,Y 567.922,Z 551.906,A -85,B 0,C 180,E1 27355.355,E2 27355.355} C_VEL
LIN {X 0,Y 567.942,Z 546.718,A -85,B 0,C 180,E1 27353.429,E2 27353.429} C_VEL
LIN {X 0,Y 567.977,Z 540.296,A -85,B 0,C 180,E1 27351.7,E2 27351.7} C_VEL
LIN {X 0,Y 568.057,Z 532.162,A -85,B 0,C 180,E1 27349.965,E2 27349.965} C_VEL
LIN {X 0,Y 568.171,Z 522.561,A -85,B 0,C 180,E1 27348.324,E2 27348.324} C_VEL
LIN {X 0,Y 568.327,Z 511.695,A -85,B 0,C 180,E1 27346.779,E2 27346.779} C_VEL
LIN {X 0,Y 568.536,Z 499.183,A -85,B 0,C 180,E1 27345.299,E2 27345.299} C_VEL
LIN {X 0,Y 568.774,Z 485.881,A -85,B 0,C 180,E1 27343.979,E2 27343.979} C_VEL
LIN {X 0,Y 569.073,Z 470.112,A -85,B 0,C 180,E1 27342.674,E2 27342.674} C_VEL
LIN {X 0,Y 569.385,Z 453.993,A -85,B 0,C 180,E1 27341.574,E2 27341.574} C_VEL
LIN {X 0,Y 569.669,Z 437.221,A -85,B 0,C 180,E1 27340.653,E2 27340.653} C_VEL
LIN {X 0,Y 569.958,Z 419.848,A -85,B 0,C 180,E1 27339.889,E2 27339.889} C_VEL
LIN {X 0,Y 570.173,Z 401.862,A -85,B 0,C 180,E1 27339.301,E2 27339.301} C_VEL
LIN {X 0,Y 570.362,Z 382.31,A -85,B 0,C 180,E1 27338.863,E2 27338.863} C_VEL
LIN {X 0,Y 570.886,Z 180.226,A -85,B 0,C 180,E1 27336.166,E2 27336.166} C_VEL
LIN {X 0,Y 570.06,Z 175.093,A -85,B 0,C 180,E1 27336.038,E2 27336.038} C_VEL
LIN {X 0,Y 570.413,Z 144.512,A -85,B 0,C 180,E1 27333.674,E2 27333.674} C_VEL
LIN {X 0,Y 570.41,Z 111.791,A -85,B 0,C 180,E1 27331.216,E2 27331.216} C_VEL
LIN {X 0,Y 570.308,Z 106.324,A -85,B 0,C 180,E1 27330.82,E2 27330.82} C_VEL
LIN {X 0,Y 568.186,Z 98.709,A -85,B 0,C 180,E1 27330.176,E2 27330.176} C_VEL
LIN {X 0,Y 568.186,Z 98.71,A -85,B 0,C 180,E1 27326.82,E2 27326.82} C_VEL
LIN {X 0,Y 568.219,Z 98.707,A -85,B 0,C 180,E1 27323.63,E2 27323.63} C_VEL
LIN {X 0,Y 568.164,Z 98.708,A -85,B 0,C 180,E1 27320.426,E2 27320.426} C_VEL
LIN {X 0,Y 568.18,Z 98.711,A -85,B 0,C 180,E1 27317.208,E2 27317.208} C_VEL
LIN {X 0,Y 568.175,Z 98.71,A -85,B 0,C 180,E1 27314.112,E2 27314.112} C_VEL
LIN {X 0,Y 568.142,Z 98.711,A -85,B 0,C 180,E1 27310.895,E2 27310.895} C_VEL
LIN {X 0,Y 568.214,Z 98.71,A -85,B 0,C 180,E1 27307.761,E2 27307.761} C_VEL
LIN {X 0,Y 568.165,Z 98.713,A -85,B 0,C 180,E1 27304.555,E2 27304.555} C_VEL
LIN {X 0,Y 568.24,Z 98.911,A -85,B 0,C 180,E1 27304.025,E2 27304.025} C_VEL
LIN {X 0,Y 572.481,Z 110.542,A -85,B 0,C 180,E1 27302.966,E2 27302.966} C_VEL
LIN {X 0,Y 571.732,Z 157.514,A -85,B 0,C 180,E1 27299.954,E2 27299.954} C_VEL
LIN {X 0,Y 571.759,Z 163.574,A -85,B 0,C 180,E1 27299.599,E2 27299.599} C_VEL
LIN {X 0,Y 572.693,Z 170.74,A -85,B 0,C 180,E1 27299.445,E2 27299.445} C_VEL
LIN {X 0,Y 571.696,Z 409.602,A -85,B 0,C 180,E1 27296.177,E2 27296.177} C_VEL
LIN {X 0,Y 571.527,Z 432.033,A -85,B 0,C 180,E1 27295.801,E2 27295.801} C_VEL
LIN {X 0,Y 571.233,Z 452.995,A -85,B 0,C 180,E1 27295.257,E2 27295.257} C_VEL
LIN {X 0,Y 570.935,Z 472.13,A -85,B 0,C 180,E1 27294.578,E2 27294.578} C_VEL
LIN {X 0,Y 570.562,Z 491.206,A -85,B 0,C 180,E1 27293.715,E2 27293.715} C_VEL
LIN {X 0,Y 570.133,Z 510.294,A -85,B 0,C 180,E1 27292.641,E2 27292.641} C_VEL
LIN {X 0,Y 569.725,Z 527.638,A -85,B 0,C 180,E1 27291.464,E2 27291.464} C_VEL
LIN {X 0,Y 569.326,Z 544.822,A -85,B 0,C 180,E1 27290.081,E2 27290.081} C_VEL
LIN {X 0,Y 568.949,Z 561.438,A -85,B 0,C 180,E1 27288.495,E2 27288.495} C_VEL
LIN {X 0,Y 568.64,Z 575.898,A -85,B 0,C 180,E1 27286.866,E2 27286.866} C_VEL
LIN {X 0,Y 568.408,Z 588.562,A -85,B 0,C 180,E1 27285.195,E2 27285.195} C_VEL
LIN {X 0,Y 568.212,Z 600.526,A -85,B 0,C 180,E1 27283.328,E2 27283.328} C_VEL
LIN {X 0,Y 568.078,Z 610.907,A -85,B 0,C 180,E1 27281.37,E2 27281.37} C_VEL
LIN {X 0,Y 567.989,Z 619.278,A -85,B 0,C 180,E1 27279.423,E2 27279.423} C_VEL
LIN {X 0,Y 567.937,Z 626.2,A -85,B 0,C 180,E1 27277.385,E2 27277.385} C_VEL
LIN {X 0,Y 567.914,Z 631.554,A -85,B 0,C 180,E1 27275.253,E2 27275.253} C_VEL
LIN {X 0,Y 567.908,Z 634.942,A -85,B 0,C 180,E1 27273.23,E2 27273.23} C_VEL
LIN {X 0,Y 567.91,Z 636.759,A -85,B 0,C 180,E1 27271.11,E2 27271.11} C_VEL
LIN {X 0,Y 567.914,Z 636.784,A -85,B 0,C 180,E1 27268.992,E2 27268.992} C_VEL
LIN {X 0,Y 567.914,Z 635.17,A -85,B 0,C 180,E1 27266.973,E2 27266.973} C_VEL
LIN {X 0,Y 567.916,Z 631.761,A -85,B 0,C 180,E1 27264.849,E2 27264.849} C_VEL
LIN {X 0,Y 567.938,Z 626.811,A -85,B 0,C 180,E1 27262.82,E2 27262.82} C_VEL
LIN {X 0,Y 567.987,Z 620.492,A -85,B 0,C 180,E1 27260.885,E2 27260.885} C_VEL
LIN {X 0,Y 568.06,Z 612.337,A -85,B 0,C 180,E1 27258.94,E2 27258.94} C_VEL
LIN {X 0,Y 568.166,Z 602.843,A -85,B 0,C 180,E1 27257.086,E2 27257.086} C_VEL
LIN {X 0,Y 568.349,Z 591.396,A -85,B 0,C 180,E1 27255.222,E2 27255.222} C_VEL
LIN {X 0,Y 568.585,Z 578.451,A -85,B 0,C 180,E1 27253.449,E2 27253.449} C_VEL
LIN {X 0,Y 568.889,Z 563.98,A -85,B 0,C 180,E1 27251.77,E2 27251.77} C_VEL
LIN {X 0,Y 569.247,Z 548.457,A -85,B 0,C 180,E1 27250.239,E2 27250.239} C_VEL
LIN {X 0,Y 569.658,Z 531.285,A -85,B 0,C 180,E1 27248.804,E2 27248.804} C_VEL
LIN {X 0,Y 570.088,Z 512.911,A -85,B 0,C 180,E1 27247.522,E2 27247.522} C_VEL
LIN {X 0,Y 570.486,Z 494.124,A -85,B 0,C 180,E1 27246.438,E2 27246.438} C_VEL
LIN {X 0,Y 570.867,Z 474.728,A -85,B 0,C 180,E1 27245.53,E2 27245.53} C_VEL
LIN {X 0,Y 571.222,Z 454.089,A -85,B 0,C 180,E1 27244.778,E2 27244.778} C_VEL
LIN {X 0,Y 571.518,Z 433.4,A -85,B 0,C 180,E1 27244.228,E2 27244.228} C_VEL
LIN {X 0,Y 571.686,Z 412.34,A -85,B 0,C 180,E1 27243.86,E2 27243.86} C_VEL
LIN {X 0,Y 572.679,Z 173.154,A -85,B 0,C 180,E1 27240.588,E2 27240.588} C_VEL
LIN {X 0,Y 572.404,Z 167.387,A -85,B 0,C 180,E1 27240.491,E2 27240.491} C_VEL
LIN {X 0,Y 571.651,Z 162.729,A -85,B 0,C 180,E1 27240.376,E2 27240.376} C_VEL
LIN {X 0,Y 572.368,Z 116.063,A -85,B 0,C 180,E1 27237.391,E2 27237.391} C_VEL
LIN {X 0,Y 572.356,Z 109.753,A -85,B 0,C 180,E1 27236.974,E2 27236.974} C_VEL
LIN {X 0,Y 568.223,Z 98.708,A -85,B 0,C 180,E1 27235.948,E2 27235.948} C_VEL
LIN {X 0,Y 568.171,Z 98.709,A -85,B 0,C 180,E1 27232.746,E2 27232.746} C_VEL
LIN {X 0,Y 568.166,Z 98.708,A -85,B 0,C 180,E1 27229.33,E2 27229.33} C_VEL
LIN {X 0,Y 568.223,Z 98.707,A -85,B 0,C 180,E1 27226.11,E2 27226.11} C_VEL
LIN {X 0,Y 568.161,Z 98.705,A -85,B 0,C 180,E1 27222.925,E2 27222.925} C_VEL
LIN {X 0,Y 568.171,Z 98.699,A -85,B 0,C 180,E1 27219.571,E2 27219.571} C_VEL
LIN {X 0,Y 568.198,Z 98.701,A -85,B 0,C 180,E1 27216.47,E2 27216.47} C_VEL
LIN {X 0,Y 568.156,Z 98.705,A -85,B 0,C 180,E1 27213.29,E2 27213.29} C_VEL
LIN {X 0,Y 568.218,Z 98.708,A -85,B 0,C 180,E1 27210.099,E2 27210.099} C_VEL
LIN {X 0,Y 568.16,Z 98.707,A -85,B 0,C 180,E1 27207.003,E2 27207.003} C_VEL
LIN {X 0,Y 568.166,Z 98.707,A -85,B 0,C 180,E1 27203.655,E2 27203.655} C_VEL
LIN {X 0,Y 568.195,Z 98.707,A -85,B 0,C 180,E1 27200.585,E2 27200.585} C_VEL
LIN {X 0,Y 568.153,Z 98.707,A -85,B 0,C 180,E1 27197.408,E2 27197.408} C_VEL
LIN {X 0,Y 568.22,Z 98.705,A -85,B 0,C 180,E1 27194.261,E2 27194.261} C_VEL
LIN {X 0,Y 568.152,Z 98.708,A -85,B 0,C 180,E1 27191.162,E2 27191.162} C_VEL
LIN {X 0,Y 568.172,Z 98.704,A -85,B 0,C 180,E1 27187.889,E2 27187.889} C_VEL
LIN {X 0,Y 568.175,Z 98.707,A -85,B 0,C 180,E1 27184.845,E2 27184.845} C_VEL
LIN {X 0,Y 568.15,Z 98.704,A -85,B 0,C 180,E1 27181.613,E2 27181.613} C_VEL
LIN {X 0,Y 568.216,Z 98.707,A -85,B 0,C 180,E1 27178.487,E2 27178.487} C_VEL
LIN {X 0,Y 568.146,Z 98.705,A -85,B 0,C 180,E1 27175.356,E2 27175.356} C_VEL
LIN {X 0,Y 568.179,Z 98.71,A -85,B 0,C 180,E1 27172.11,E2 27172.11} C_VEL
LIN {X 0,Y 568.163,Z 98.706,A -85,B 0,C 180,E1 27169.044,E2 27169.044} C_VEL
LIN {X 0,Y 568.148,Z 98.709,A -85,B 0,C 180,E1 27165.736,E2 27165.736} C_VEL
LIN {X 0,Y 568.212,Z 98.705,A -85,B 0,C 180,E1 27162.594,E2 27162.594} C_VEL
LIN {X 0,Y 568.148,Z 98.709,A -85,B 0,C 180,E1 27159.825,E2 27159.825} C_VEL
LIN {X 0,Y 567.162,Z 98.835,A -85,B 0,C 180,E1 27159.049,E2 27159.049} C_VEL
LIN {X 0,Y 560.714,Z 99.644,A -85,B 0,C 180,E1 27156.811,E2 27156.811} C_VEL
LIN {X 0,Y 560.244,Z 99.697,A -85,B 0,C 180,E1 27156.3,E2 27156.3} C_VEL
LIN {X 0,Y 560.221,Z 99.698,A -85,B 0,C 180,E1 27153.157,E2 27153.157} C_VEL
LIN {X 0,Y 560.206,Z 99.698,A -85,B 0,C 180,E1 27149.898,E2 27149.898} C_VEL
LIN {X 0,Y 560.262,Z 99.695,A -85,B 0,C 180,E1 27146.778,E2 27146.778} C_VEL
LIN {X 0,Y 560.201,Z 99.698,A -85,B 0,C 180,E1 27143.604,E2 27143.604} C_VEL
LIN {X 0,Y 560.241,Z 99.698,A -85,B 0,C 180,E1 27140.421,E2 27140.421} C_VEL
LIN {X 0,Y 560.212,Z 99.699,A -85,B 0,C 180,E1 27137.334,E2 27137.334} C_VEL
LIN {X 0,Y 560.203,Z 99.7,A -85,B 0,C 180,E1 27133.97,E2 27133.97} C_VEL
LIN {X 0,Y 560.272,Z 99.698,A -85,B 0,C 180,E1 27130.779,E2 27130.779} C_VEL
LIN {X 0,Y 560.202,Z 99.698,A -85,B 0,C 180,E1 27127.618,E2 27127.618} C_VEL
LIN {X 0,Y 560.218,Z 99.702,A -85,B 0,C 180,E1 27124.274,E2 27124.274} C_VEL
LIN {X 0,Y 560.232,Z 99.703,A -85,B 0,C 180,E1 27121.253,E2 27121.253} C_VEL
LIN {X 0,Y 560.271,Z 99.804,A -85,B 0,C 180,E1 27120.663,E2 27120.663} C_VEL
LIN {X 0,Y 564.034,Z 111.268,A -85,B 0,C 180,E1 27119.446,E2 27119.446} C_VEL
LIN {X 0,Y 563.214,Z 149.659,A -85,B 0,C 180,E1 27116.296,E2 27116.296} C_VEL
LIN {X 0,Y 562.746,Z 175.55,A -85,B 0,C 180,E1 27114.238,E2 27114.238} C_VEL
LIN {X 0,Y 563.892,Z 183.772,A -85,B 0,C 180,E1 27114.065,E2 27114.065} C_VEL
LIN {X 0,Y 562.882,Z 384.656,A -85,B 0,C 180,E1 27111.303,E2 27111.303} C_VEL
LIN {X 0,Y 562.656,Z 403.571,A -85,B 0,C 180,E1 27110.852,E2 27110.852} C_VEL
LIN {X 0,Y 562.373,Z 421.631,A -85,B 0,C 180,E1 27110.23,E2 27110.23} C_VEL
LIN {X 0,Y 562.023,Z 439.214,A -85,B 0,C 180,E1 27109.431,E2 27109.431} C_VEL
LIN {X 0,Y 561.665,Z 455.908,A -85,B 0,C 180,E1 27108.473,E2 27108.473} C_VEL
LIN {X 0,Y 561.306,Z 471.738,A -85,B 0,C 180,E1 27107.359,E2 27107.359} C_VEL
LIN {X 0,Y 560.964,Z 486.404,A -85,B 0,C 180,E1 27106.113,E2 27106.113} C_VEL
LIN {X 0,Y 560.651,Z 500.557,A -85,B 0,C 180,E1 27104.669,E2 27104.669} C_VEL
LIN {X 0,Y 560.393,Z 513.36,A -85,B 0,C 180,E1 27103.096,E2 27103.096} C_VEL
LIN {X 0,Y 560.194,Z 524.596,A -85,B 0,C 180,E1 27101.426,E2 27101.426} C_VEL
LIN {X 0,Y 560.06,Z 534.288,A -85,B 0,C 180,E1 27099.66,E2 27099.66} C_VEL
LIN {X 0,Y 559.982,Z 542.005,A -85,B 0,C 180,E1 27097.902,E2 27097.902} C_VEL
LIN {X 0,Y 559.938,Z 548.285,A -85,B 0,C 180,E1 27096.047,E2 27096.047} C_VEL
LIN {X 0,Y 559.919,Z 552.788,A -85,B 0,C 180,E1 27094.198,E2 27094.198} C_VEL
LIN {X 0,Y 559.914,Z 555.744,A -85,B 0,C 180,E1 27092.251,E2 27092.251} C_VEL
LIN {X 0,Y 559.909,Z 556.93,A -85,B 0,C 180,E1 27090.306,E2 27090.306} C_VEL
LIN {X 0,Y 559.914,Z 556.377,A -85,B 0,C 180,E1 27088.362,E2 27088.362} C_VEL
LIN {X 0,Y 559.909,Z 554.072,A -85,B 0,C 180,E1 27086.416,E2 27086.416} C_VEL
LIN {X 0,Y 559.928,Z 550.206,A -85,B 0,C 180,E1 27084.569,E2 27084.569} C_VEL
LIN {X 0,Y 559.954,Z 544.618,A -85,B 0,C 180,E1 27082.716,E2 27082.716} C_VEL
LIN {X 0,Y 560.033,Z 537.184,A -85,B 0,C 180,E1 27080.861,E2 27080.861} C_VEL
LIN {X 0,Y 560.142,Z 528.186,A -85,B 0,C 180,E1 27079.093,E2 27079.093} C_VEL
LIN {X 0,Y 560.317,Z 517.746,A -85,B 0,C 180,E1 27077.425,E2 27077.425} C_VEL
LIN {X 0,Y 560.543,Z 505.86,A -85,B 0,C 180,E1 27075.855,E2 27075.855} C_VEL
LIN {X 0,Y 560.83,Z 492.491,A -85,B 0,C 180,E1 27074.382,E2 27074.382} C_VEL
LIN {X 0,Y 561.174,Z 477.497,A -85,B 0,C 180,E1 27073.01,E2 27073.01} C_VEL
LIN {X 0,Y 561.543,Z 461.342,A -85,B 0,C 180,E1 27071.793,E2 27071.793} C_VEL
LIN {X 0,Y 561.906,Z 444.883,A -85,B 0,C 180,E1 27070.78,E2 27070.78} C_VEL
LIN {X 0,Y 562.262,Z 427.586,A -85,B 0,C 180,E1 27069.927,E2 27069.927} C_VEL
LIN {X 0,Y 562.572,Z 409.273,A -85,B 0,C 180,E1 27069.234,E2 27069.234} C_VEL
LIN {X 0,Y 562.817,Z 390.814,A -85,B 0,C 180,E1 27068.734,E2 27068.734} C_VEL
LIN {X 0,Y 562.979,Z 369.896,A -85,B 0,C 180,E1 27068.38,E2 27068.38} C_VEL
LIN {X 0,Y 563.79,Z 181.552,A -85,B 0,C 180,E1 27065.81,E2 27065.81} C_VEL
LIN {X 0,Y 562.666,Z 174.963,A -85,B 0,C 180,E1 27065.652,E2 27065.652} C_VEL
LIN {X 0,Y 563.475,Z 135.601,A -85,B 0,C 180,E1 27062.467,E2 27062.467} C_VEL
LIN {X 0,Y 563.93,Z 110.706,A -85,B 0,C 180,E1 27060.41,E2 27060.41} C_VEL
LIN {X 0,Y 560.276,Z 99.699,A -85,B 0,C 180,E1 27059.22,E2 27059.22} C_VEL
LIN {X 0,Y 560.221,Z 99.699,A -85,B 0,C 180,E1 27056.038,E2 27056.038} C_VEL
LIN {X 0,Y 560.235,Z 99.698,A -85,B 0,C 180,E1 27052.641,E2 27052.641} C_VEL
LIN {X 0,Y 560.284,Z 99.694,A -85,B 0,C 180,E1 27049.484,E2 27049.484} C_VEL
LIN {X 0,Y 560.265,Z 99.695,A -85,B 0,C 180,E1 27046.136,E2 27046.136} C_VEL
LIN {X 0,Y 560.26,Z 99.691,A -85,B 0,C 180,E1 27042.82,E2 27042.82} C_VEL
LIN {X 0,Y 560.273,Z 99.692,A -85,B 0,C 180,E1 27039.561,E2 27039.561} C_VEL
LIN {X 0,Y 560.271,Z 99.698,A -85,B 0,C 180,E1 27036.207,E2 27036.207} C_VEL
LIN {X 0,Y 560.279,Z 99.697,A -85,B 0,C 180,E1 27032.803,E2 27032.803} C_VEL
LIN {X 0,Y 560.27,Z 99.833,A -85,B 0,C 180,E1 27030.306,E2 27030.306} C_VEL
LIN {X 0,Y 563.362,Z 110.042,A -85,B 0,C 180,E1 27029.331,E2 27029.331} C_VEL
LIN {X 0,Y 562.938,Z 149.98,A -85,B 0,C 180,E1 27026.197,E2 27026.197} C_VEL
LIN {X 0,Y 562.591,Z 176.303,A -85,B 0,C 180,E1 27024.152,E2 27024.152} C_VEL
LIN {X 0,Y 563.596,Z 183.925,A -85,B 0,C 180,E1 27024.005,E2 27024.005} C_VEL
LIN {X 0,Y 562.888,Z 383.615,A -85,B 0,C 180,E1 27021.319,E2 27021.319} C_VEL
LIN {X 0,Y 562.665,Z 402.316,A -85,B 0,C 180,E1 27020.883,E2 27020.883} C_VEL
LIN {X 0,Y 562.398,Z 420.315,A -85,B 0,C 180,E1 27020.285,E2 27020.285} C_VEL
LIN {X 0,Y 562.053,Z 437.012,A -85,B 0,C 180,E1 27019.539,E2 27019.539} C_VEL
LIN {X 0,Y 561.699,Z 454.186,A -85,B 0,C 180,E1 27018.58,E2 27018.58} C_VEL
LIN {X 0,Y 561.34,Z 470.113,A -85,B 0,C 180,E1 27017.484,E2 27017.484} C_VEL
LIN {X 0,Y 560.974,Z 485.448,A -85,B 0,C 180,E1 27016.197,E2 27016.197} C_VEL
LIN {X 0,Y 560.695,Z 498.146,A -85,B 0,C 180,E1 27014.933,E2 27014.933} C_VEL
LIN {X 0,Y 560.434,Z 510.983,A -85,B 0,C 180,E1 27013.411,E2 27013.411} C_VEL
LIN {X 0,Y 560.246,Z 521.297,A -85,B 0,C 180,E1 27011.948,E2 27011.948} C_VEL
LIN {X 0,Y 560.103,Z 531.15,A -85,B 0,C 180,E1 27010.283,E2 27010.283} C_VEL
LIN {X 0,Y 560.007,Z 539.476,A -85,B 0,C 180,E1 27008.522,E2 27008.522} C_VEL
LIN {X 0,Y 559.953,Z 546.078,A -85,B 0,C 180,E1 27006.768,E2 27006.768} C_VEL
LIN {X 0,Y 559.918,Z 551.47,A -85,B 0,C 180,E1 27004.815,E2 27004.815} C_VEL
LIN {X 0,Y 559.914,Z 554.712,A -85,B 0,C 180,E1 27003.071,E2 27003.071} C_VEL
LIN {X 0,Y 559.907,Z 556.705,A -85,B 0,C 180,E1 27001.023,E2 27001.023} C_VEL
LIN {X 0,Y 559.912,Z 556.809,A -85,B 0,C 180,E1 26999.182,E2 26999.182} C_VEL
LIN {X 0,Y 559.909,Z 555.289,A -85,B 0,C 180,E1 26997.237,E2 26997.237} C_VEL
LIN {X 0,Y 559.922,Z 552.115,A -85,B 0,C 180,E1 26995.391,E2 26995.391} C_VEL
LIN {X 0,Y 559.945,Z 547.355,A -85,B 0,C 180,E1 26993.541,E2 26993.541} C_VEL
LIN {X 0,Y 559.989,Z 540.709,A -85,B 0,C 180,E1 26991.685,E2 26991.685} C_VEL
LIN {X 0,Y 560.083,Z 532.679,A -85,B 0,C 180,E1 26989.924,E2 26989.924} C_VEL
LIN {X 0,Y 560.232,Z 522.546,A -85,B 0,C 180,E1 26988.156,E2 26988.156} C_VEL
LIN {X 0,Y 560.424,Z 511.69,A -85,B 0,C 180,E1 26986.589,E2 26986.589} C_VEL
LIN {X 0,Y 560.688,Z 498.475,A -85,B 0,C 180,E1 26985.015,E2 26985.015} C_VEL
LIN {X 0,Y 560.984,Z 485.309,A -85,B 0,C 180,E1 26983.697,E2 26983.697} C_VEL
LIN {X 0,Y 561.345,Z 469.376,A -85,B 0,C 180,E1 26982.374,E2 26982.374} C_VEL
LIN {X 0,Y 561.708,Z 453.974,A -85,B 0,C 180,E1 26981.313,E2 26981.313} C_VEL
LIN {X 0,Y 562.048,Z 437.626,A -85,B 0,C 180,E1 26980.403,E2 26980.403} C_VEL
LIN {X 0,Y 562.397,Z 420.549,A -85,B 0,C 180,E1 26979.634,E2 26979.634} C_VEL
LIN {X 0,Y 562.655,Z 402.494,A -85,B 0,C 180,E1 26979.032,E2 26979.032} C_VEL
LIN {X 0,Y 562.885,Z 383.582,A -85,B 0,C 180,E1 26978.591,E2 26978.591} C_VEL
LIN {X 0,Y 563.211,Z 285.222,A -85,B 0,C 180,E1 26977.268,E2 26977.268} C_VEL
LIN {X 0,Y 563.381,Z 180.938,A -85,B 0,C 180,E1 26975.872,E2 26975.872} C_VEL
LIN {X 0,Y 562.609,Z 176.008,A -85,B 0,C 180,E1 26975.741,E2 26975.741} C_VEL
LIN {X 0,Y 562.941,Z 141.96,A -85,B 0,C 180,E1 26973.121,E2 26973.121} C_VEL
LIN {X 0,Y 562.819,Z 108.819,A -85,B 0,C 180,E1 26970.668,E2 26970.668} C_VEL
LIN {X 0,Y 560.263,Z 99.697,A -85,B 0,C 180,E1 26969.902,E2 26969.902} C_VEL
LIN {X 0,Y 560.239,Z 99.698,A -85,B 0,C 180,E1 26966.641,E2 26966.641} C_VEL
LIN {X 0,Y 560.284,Z 99.698,A -85,B 0,C 180,E1 26963.413,E2 26963.413} C_VEL
LIN {X 0,Y 560.23,Z 99.697,A -85,B 0,C 180,E1 26960.284,E2 26960.284} C_VEL
LIN {X 0,Y 560.219,Z 99.699,A -85,B 0,C 180,E1 26956.877,E2 26956.877} C_VEL
LIN {X 0,Y 560.276,Z 99.699,A -85,B 0,C 180,E1 26953.681,E2 26953.681} C_VEL
LIN {X 0,Y 560.208,Z 99.701,A -85,B 0,C 180,E1 26950.507,E2 26950.507} C_VEL
LIN {X 0,Y 560.214,Z 99.701,A -85,B 0,C 180,E1 26947.08,E2 26947.08} C_VEL
LIN {X 0,Y 560.258,Z 99.9,A -85,B 0,C 180,E1 26944.493,E2 26944.493} C_VEL
LIN {X 0,Y 565.433,Z 113.411,A -85,B 0,C 180,E1 26943.237,E2 26943.237} C_VEL
LIN {X 0,Y 564.524,Z 160.295,A -85,B 0,C 180,E1 26940.195,E2 26940.195} C_VEL
LIN {X 0,Y 564.597,Z 163.654,A -85,B 0,C 180,E1 26940.012,E2 26940.012} C_VEL
LIN {X 0,Y 565.718,Z 172,A -85,B 0,C 180,E1 26939.826,E2 26939.826} C_VEL
LIN {X 0,Y 564.51,Z 411.094,A -85,B 0,C 180,E1 26936.515,E2 26936.515} C_VEL
LIN {X 0,Y 564.305,Z 432.681,A -85,B 0,C 180,E1 26936.141,E2 26936.141} C_VEL
LIN {X 0,Y 563.948,Z 453.785,A -85,B 0,C 180,E1 26935.581,E2 26935.581} C_VEL
LIN {X 0,Y 563.563,Z 473.412,A -85,B 0,C 180,E1 26934.865,E2 26934.865} C_VEL
LIN {X 0,Y 563.12,Z 492.261,A -85,B 0,C 180,E1 26933.992,E2 26933.992} C_VEL
LIN {X 0,Y 562.611,Z 511.188,A -85,B 0,C 180,E1 26932.905,E2 26932.905} C_VEL
LIN {X 0,Y 562.099,Z 529.095,A -85,B 0,C 180,E1 26931.661,E2 26931.661} C_VEL
LIN {X 0,Y 561.636,Z 545.428,A -85,B 0,C 180,E1 26930.314,E2 26930.314} C_VEL
LIN {X 0,Y 561.191,Z 561.43,A -85,B 0,C 180,E1 26928.761,E2 26928.761} C_VEL
LIN {X 0,Y 560.814,Z 575.899,A -85,B 0,C 180,E1 26927.109,E2 26927.109} C_VEL
LIN {X 0,Y 560.525,Z 588.564,A -85,B 0,C 180,E1 26925.414,E2 26925.414} C_VEL
LIN {X 0,Y 560.279,Z 600.527,A -85,B 0,C 180,E1 26923.52,E2 26923.52} C_VEL
LIN {X 0,Y 560.111,Z 610.906,A -85,B 0,C 180,E1 26921.534,E2 26921.534} C_VEL
LIN {X 0,Y 560.005,Z 619.277,A -85,B 0,C 180,E1 26919.559,E2 26919.559} C_VEL
LIN {X 0,Y 559.945,Z 626.2,A -85,B 0,C 180,E1 26917.491,E2 26917.491} C_VEL
LIN {X 0,Y 559.916,Z 631.348,A -85,B 0,C 180,E1 26915.431,E2 26915.431} C_VEL
LIN {X 0,Y 559.906,Z 634.828,A -85,B 0,C 180,E1 26913.379,E2 26913.379} C_VEL
LIN {X 0,Y 559.907,Z 636.706,A -85,B 0,C 180,E1 26911.229,E2 26911.229} C_VEL
LIN {X 0,Y 559.91,Z 636.829,A -85,B 0,C 180,E1 26909.182,E2 26909.182} C_VEL
LIN {X 0,Y 559.915,Z 635.282,A -85,B 0,C 180,E1 26907.032,E2 26907.032} C_VEL
LIN {X 0,Y 559.919,Z 631.966,A -85,B 0,C 180,E1 26904.878,E2 26904.878} C_VEL
LIN {X 0,Y 559.943,Z 627.114,A -85,B 0,C 180,E1 26902.82,E2 26902.82} C_VEL
LIN {X 0,Y 560,Z 620.492,A -85,B 0,C 180,E1 26900.754,E2 26900.754} C_VEL
LIN {X 0,Y 560.096,Z 612.338,A -85,B 0,C 180,E1 26898.78,E2 26898.78} C_VEL
LIN {X 0,Y 560.236,Z 602.844,A -85,B 0,C 180,E1 26896.9,E2 26896.9} C_VEL
LIN {X 0,Y 560.457,Z 591.396,A -85,B 0,C 180,E1 26895.009,E2 26895.009} C_VEL
LIN {X 0,Y 560.745,Z 578.451,A -85,B 0,C 180,E1 26893.211,E2 26893.211} C_VEL
LIN {X 0,Y 561.103,Z 564.699,A -85,B 0,C 180,E1 26891.584,E2 26891.584} C_VEL
LIN {X 0,Y 561.536,Z 549.059,A -85,B 0,C 180,E1 26890.01,E2 26890.01} C_VEL
LIN {X 0,Y 562.026,Z 531.964,A -85,B 0,C 180,E1 26888.557,E2 26888.557} C_VEL
LIN {X 0,Y 562.531,Z 514.213,A -85,B 0,C 180,E1 26887.292,E2 26887.292} C_VEL
LIN {X 0,Y 562.994,Z 496.3,A -85,B 0,C 180,E1 26886.226,E2 26886.226} C_VEL
LIN {X 0,Y 563.473,Z 476.716,A -85,B 0,C 180,E1 26885.275,E2 26885.275} C_VEL
LIN {X 0,Y 563.914,Z 456.684,A -85,B 0,C 180,E1 26884.512,E2 26884.512} C_VEL
LIN {X 0,Y 564.277,Z 436.445,A -85,B 0,C 180,E1 26883.939,E2 26883.939} C_VEL
LIN {X 0,Y 564.484,Z 415.387,A -85,B 0,C 180,E1 26883.545,E2 26883.545} C_VEL
LIN {X 0,Y 565.683,Z 177.588,A -85,B 0,C 180,E1 26880.252,E2 26880.252} C_VEL
LIN {X 0,Y 565.489,Z 168.968,A -85,B 0,C 180,E1 26880.117,E2 26880.117} C_VEL
LIN {X 0,Y 564.481,Z 162.496,A -85,B 0,C 180,E1 26879.946,E2 26879.946} C_VEL
LIN {X 0,Y 565.368,Z 116.065,A -85,B 0,C 180,E1 26876.936,E2 26876.936} C_VEL
LIN {X 0,Y 565.279,Z 112.68,A -85,B 0,C 180,E1 26876.703,E2 26876.703} C_VEL
LIN {X 0,Y 560.24,Z 99.702,A -85,B 0,C 180,E1 26875.474,E2 26875.474} C_VEL
LIN {X 0,Y 560.278,Z 99.697,A -85,B 0,C 180,E1 26872.238,E2 26872.238} C_VEL
LIN {X 0,Y 560.222,Z 99.696,A -85,B 0,C 180,E1 26869.021,E2 26869.021} C_VEL
LIN {X 0,Y 560.251,Z 99.699,A -85,B 0,C 180,E1 26865.696,E2 26865.696} C_VEL
LIN {X 0,Y 560.249,Z 99.693,A -85,B 0,C 180,E1 26862.519,E2 26862.519} C_VEL
LIN {X 0,Y 560.22,Z 99.686,A -85,B 0,C 180,E1 26859.315,E2 26859.315} C_VEL
LIN {X 0,Y 560.278,Z 99.693,A -85,B 0,C 180,E1 26856.079,E2 26856.079} C_VEL
LIN {X 0,Y 560.222,Z 99.693,A -85,B 0,C 180,E1 26852.98,E2 26852.98} C_VEL
LIN {X 0,Y 560.232,Z 99.695,A -85,B 0,C 180,E1 26849.628,E2 26849.628} C_VEL
LIN {X 0,Y 560.261,Z 99.695,A -85,B 0,C 180,E1 26846.497,E2 26846.497} C_VEL
LIN {X 0,Y 560.216,Z 99.694,A -85,B 0,C 180,E1 26843.342,E2 26843.342} C_VEL
LIN {X 0,Y 560.272,Z 99.695,A -85,B 0,C 180,E1 26840.147,E2 26840.147} C_VEL
LIN {X 0,Y 560.226,Z 99.695,A -85,B 0,C 180,E1 26836.941,E2 26836.941} C_VEL
LIN {X 0,Y 560.22,Z 99.692,A -85,B 0,C 180,E1 26833.626,E2 26833.626} C_VEL
LIN {X 0,Y 560.282,Z 99.696,A -85,B 0,C 180,E1 26830.384,E2 26830.384} C_VEL
LIN {X 0,Y 560.215,Z 99.691,A -85,B 0,C 180,E1 26827.177,E2 26827.177} C_VEL
LIN {X 0,Y 560.223,Z 99.698,A -85,B 0,C 180,E1 26823.786,E2 26823.786} C_VEL
LIN {X 0,Y 560.265,Z 99.691,A -85,B 0,C 180,E1 26820.613,E2 26820.613} C_VEL
LIN {X 0,Y 560.209,Z 99.698,A -85,B 0,C 180,E1 26817.442,E2 26817.442} C_VEL
LIN {X 0,Y 560.26,Z 99.694,A -85,B 0,C 180,E1 26814.264,E2 26814.264} C_VEL
LIN {X 0,Y 560.217,Z 99.698,A -85,B 0,C 180,E1 26811.171,E2 26811.171} C_VEL
LIN {X 0,Y 560.215,Z 99.695,A -85,B 0,C 180,E1 26807.842,E2 26807.842} C_VEL
LIN {X 0,Y 560.267,Z 99.698,A -85,B 0,C 180,E1 26804.685,E2 26804.685} C_VEL
LIN {X 0,Y 560.205,Z 99.695,A -85,B 0,C 180,E1 26801.476,E2 26801.476} C_VEL
LIN {X 0,Y 560.235,Z 99.696,A -85,B 0,C 180,E1 26798.209,E2 26798.209} C_VEL
LIN {X 0,Y 560.244,Z 99.697,A -85,B 0,C 180,E1 26796.3,E2 26796.3} C_VEL
LIN {X 0,Y 559.208,Z 99.822,A -85,B 0,C 180,E1 26795.513,E2 26795.513} C_VEL
LIN {X 0,Y 552.838,Z 100.631,A -85,B 0,C 180,E1 26793.301,E2 26793.301} C_VEL
LIN {X 0,Y 552.327,Z 100.686,A -85,B 0,C 180,E1 26792.726,E2 26792.726} C_VEL
LIN {X 0,Y 552.264,Z 100.687,A -85,B 0,C 180,E1 26789.516,E2 26789.516} C_VEL
LIN {X 0,Y 552.285,Z 100.687,A -85,B 0,C 180,E1 26786.197,E2 26786.197} C_VEL
LIN {X 0,Y 552.294,Z 100.687,A -85,B 0,C 180,E1 26783.055,E2 26783.055} C_VEL
LIN {X 0,Y 552.262,Z 100.687,A -85,B 0,C 180,E1 26779.819,E2 26779.819} C_VEL
LIN {X 0,Y 552.325,Z 100.686,A -85,B 0,C 180,E1 26776.678,E2 26776.678} C_VEL
LIN {X 0,Y 552.266,Z 100.689,A -85,B 0,C 180,E1 26773.469,E2 26773.469} C_VEL
LIN {X 0,Y 552.264,Z 100.688,A -85,B 0,C 180,E1 26770.019,E2 26770.019} C_VEL
LIN {X 0,Y 552.331,Z 100.688,A -85,B 0,C 180,E1 26766.857,E2 26766.857} C_VEL
LIN {X 0,Y 552.267,Z 100.691,A -85,B 0,C 180,E1 26763.611,E2 26763.611} C_VEL
LIN {X 0,Y 552.334,Z 100.861,A -85,B 0,C 180,E1 26761.102,E2 26761.102} C_VEL
LIN {X 0,Y 556.779,Z 114.386,A -85,B 0,C 180,E1 26759.638,E2 26759.638} C_VEL
LIN {X 0,Y 555.808,Z 152.946,A -85,B 0,C 180,E1 26756.437,E2 26756.437} C_VEL
LIN {X 0,Y 555.356,Z 175.464,A -85,B 0,C 180,E1 26754.631,E2 26754.631} C_VEL
LIN {X 0,Y 556.772,Z 184.801,A -85,B 0,C 180,E1 26754.428,E2 26754.428} C_VEL
LIN {X 0,Y 555.704,Z 383.803,A -85,B 0,C 180,E1 26751.682,E2 26751.682} C_VEL
LIN {X 0,Y 555.402,Z 402.819,A -85,B 0,C 180,E1 26751.227,E2 26751.227} C_VEL
LIN {X 0,Y 555.023,Z 420.242,A -85,B 0,C 180,E1 26750.62,E2 26750.62} C_VEL
LIN {X 0,Y 554.537,Z 437.726,A -85,B 0,C 180,E1 26749.814,E2 26749.814} C_VEL
LIN {X 0,Y 554.022,Z 454.929,A -85,B 0,C 180,E1 26748.803,E2 26748.803} C_VEL
LIN {X 0,Y 553.59,Z 471.076,A -85,B 0,C 180,E1 26747.663,E2 26747.663} C_VEL
LIN {X 0,Y 553.174,Z 486.097,A -85,B 0,C 180,E1 26746.377,E2 26746.377} C_VEL
LIN {X 0,Y 552.819,Z 499.636,A -85,B 0,C 180,E1 26744.988,E2 26744.988} C_VEL
LIN {X 0,Y 552.527,Z 511.822,A -85,B 0,C 180,E1 26743.499,E2 26743.499} C_VEL
LIN {X 0,Y 552.284,Z 523.328,A -85,B 0,C 180,E1 26741.804,E2 26741.804} C_VEL
LIN {X 0,Y 552.12,Z 532.747,A -85,B 0,C 180,E1 26740.116,E2 26740.116} C_VEL
LIN {X 0,Y 552.012,Z 540.792,A -85,B 0,C 180,E1 26738.331,E2 26738.331} C_VEL
LIN {X 0,Y 551.943,Z 547.377,A -85,B 0,C 180,E1 26736.448,E2 26736.448} C_VEL
LIN {X 0,Y 551.921,Z 552.17,A -85,B 0,C 180,E1 26734.571,E2 26734.571} C_VEL
LIN {X 0,Y 551.909,Z 555.29,A -85,B 0,C 180,E1 26732.699,E2 26732.699} C_VEL
LIN {X 0,Y 551.916,Z 556.839,A -85,B 0,C 180,E1 26730.726,E2 26730.726} C_VEL
LIN {X 0,Y 551.908,Z 556.646,A -85,B 0,C 180,E1 26728.754,E2 26728.754} C_VEL
LIN {X 0,Y 551.914,Z 554.707,A -85,B 0,C 180,E1 26726.78,E2 26726.78} C_VEL
LIN {X 0,Y 551.924,Z 551.22,A -85,B 0,C 180,E1 26724.907,E2 26724.907} C_VEL
LIN {X 0,Y 551.961,Z 546.027,A -85,B 0,C 180,E1 26723.028,E2 26723.028} C_VEL
LIN {X 0,Y 552.021,Z 539.453,A -85,B 0,C 180,E1 26721.248,E2 26721.248} C_VEL
LIN {X 0,Y 552.145,Z 531.051,A -85,B 0,C 180,E1 26719.461,E2 26719.461} C_VEL
LIN {X 0,Y 552.322,Z 521.247,A -85,B 0,C 180,E1 26717.771,E2 26717.771} C_VEL
LIN {X 0,Y 552.565,Z 510.082,A -85,B 0,C 180,E1 26716.181,E2 26716.181} C_VEL
LIN {X 0,Y 552.89,Z 497.046,A -85,B 0,C 180,E1 26714.636,E2 26714.636} C_VEL
LIN {X 0,Y 553.267,Z 482.973,A -85,B 0,C 180,E1 26713.246,E2 26713.246} C_VEL
LIN {X 0,Y 553.676,Z 467.985,A -85,B 0,C 180,E1 26712.012,E2 26712.012} C_VEL
LIN {X 0,Y 554.123,Z 451.331,A -85,B 0,C 180,E1 26710.882,E2 26710.882} C_VEL
LIN {X 0,Y 554.626,Z 434.274,A -85,B 0,C 180,E1 26709.925,E2 26709.925} C_VEL
LIN {X 0,Y 555.092,Z 416.399,A -85,B 0,C 180,E1 26709.144,E2 26709.144} C_VEL
LIN {X 0,Y 555.469,Z 397.635,A -85,B 0,C 180,E1 26708.542,E2 26708.542} C_VEL
LIN {X 0,Y 555.739,Z 378.502,A -85,B 0,C 180,E1 26708.141,E2 26708.141} C_VEL
LIN {X 0,Y 556.696,Z 182.921,A -85,B 0,C 180,E1 26705.456,E2 26705.456} C_VEL
LIN {X 0,Y 555.28,Z 174.767,A -85,B 0,C 180,E1 26705.25,E2 26705.25} C_VEL
LIN {X 0,Y 556.226,Z 135.329,A -85,B 0,C 180,E1 26702.019,E2 26702.019} C_VEL
LIN {X 0,Y 556.601,Z 113.526,A -85,B 0,C 180,E1 26700.187,E2 26700.187} C_VEL
LIN {X 0,Y 552.293,Z 100.692,A -85,B 0,C 180,E1 26698.756,E2 26698.756} C_VEL
LIN {X 0,Y 552.316,Z 100.689,A -85,B 0,C 180,E1 26695.61,E2 26695.61} C_VEL
LIN {X 0,Y 552.293,Z 100.689,A -85,B 0,C 180,E1 26692.292,E2 26692.292} C_VEL
LIN {X 0,Y 552.325,Z 100.683,A -85,B 0,C 180,E1 26689.016,E2 26689.016} C_VEL
LIN {X 0,Y 552.341,Z 100.685,A -85,B 0,C 180,E1 26685.647,E2 26685.647} C_VEL
LIN {X 0,Y 552.333,Z 100.685,A -85,B 0,C 180,E1 26682.235,E2 26682.235} C_VEL
LIN {X 0,Y 552.329,Z 100.682,A -85,B 0,C 180,E1 26678.884,E2 26678.884} C_VEL
LIN {X 0,Y 552.331,Z 100.682,A -85,B 0,C 180,E1 26675.528,E2 26675.528} C_VEL
LIN {X 0,Y 552.316,Z 100.688,A -85,B 0,C 180,E1 26672.156,E2 26672.156} C_VEL
LIN {X 0,Y 552.365,Z 100.875,A -85,B 0,C 180,E1 26670.665,E2 26670.665} C_VEL
LIN {X 0,Y 555.966,Z 113.044,A -85,B 0,C 180,E1 26669.49,E2 26669.49} C_VEL
LIN {X 0,Y 555.435,Z 153.608,A -85,B 0,C 180,E1 26666.285,E2 26666.285} C_VEL
LIN {X 0,Y 555.139,Z 176.784,A -85,B 0,C 180,E1 26664.48,E2 26664.48} C_VEL
LIN {X 0,Y 556.226,Z 184.992,A -85,B 0,C 180,E1 26664.313,E2 26664.313} C_VEL
LIN {X 0,Y 555.343,Z 384.835,A -85,B 0,C 180,E1 26661.576,E2 26661.576} C_VEL
LIN {X 0,Y 555.105,Z 403.395,A -85,B 0,C 180,E1 26661.133,E2 26661.133} C_VEL
LIN {X 0,Y 554.818,Z 420.899,A -85,B 0,C 180,E1 26660.541,E2 26660.541} C_VEL
LIN {X 0,Y 554.429,Z 438.055,A -85,B 0,C 180,E1 26659.764,E2 26659.764} C_VEL
LIN {X 0,Y 554.018,Z 454.787,A -85,B 0,C 180,E1 26658.808,E2 26658.808} C_VEL
LIN {X 0,Y 553.604,Z 470.643,A -85,B 0,C 180,E1 26657.697,E2 26657.697} C_VEL
LIN {X 0,Y 553.182,Z 485.441,A -85,B 0,C 180,E1 26656.432,E2 26656.432} C_VEL
LIN {X 0,Y 552.853,Z 498.142,A -85,B 0,C 180,E1 26655.15,E2 26655.15} C_VEL
LIN {X 0,Y 552.538,Z 510.982,A -85,B 0,C 180,E1 26653.606,E2 26653.606} C_VEL
LIN {X 0,Y 552.311,Z 521.29,A -85,B 0,C 180,E1 26652.122,E2 26652.122} C_VEL
LIN {X 0,Y 552.145,Z 531.155,A -85,B 0,C 180,E1 26650.433,E2 26650.433} C_VEL
LIN {X 0,Y 552.024,Z 539.469,A -85,B 0,C 180,E1 26648.647,E2 26648.647} C_VEL
LIN {X 0,Y 551.959,Z 546.081,A -85,B 0,C 180,E1 26646.867,E2 26646.867} C_VEL
LIN {X 0,Y 551.92,Z 551.236,A -85,B 0,C 180,E1 26644.989,E2 26644.989} C_VEL
LIN {X 0,Y 551.912,Z 554.55,A -85,B 0,C 180,E1 26643.22,E2 26643.22} C_VEL
LIN {X 0,Y 551.909,Z 556.616,A -85,B 0,C 180,E1 26641.246,E2 26641.246} C_VEL
LIN {X 0,Y 551.915,Z 556.856,A -85,B 0,C 180,E1 26639.377,E2 26639.377} C_VEL
LIN {X 0,Y 551.914,Z 555.64,A -85,B 0,C 180,E1 26637.508,E2 26637.508} C_VEL
LIN {X 0,Y 551.92,Z 552.54,A -85,B 0,C 180,E1 26635.532,E2 26635.532} C_VEL
LIN {X 0,Y 551.946,Z 547.96,A -85,B 0,C 180,E1 26633.656,E2 26633.656} C_VEL
LIN {X 0,Y 552.001,Z 541.121,A -85,B 0,C 180,E1 26631.668,E2 26631.668} C_VEL
LIN {X 0,Y 552.102,Z 533.695,A -85,B 0,C 180,E1 26629.988,E2 26629.988} C_VEL
LIN {X 0,Y 552.284,Z 523.198,A -85,B 0,C 180,E1 26628.09,E2 26628.09} C_VEL
LIN {X 0,Y 552.488,Z 513.211,A -85,B 0,C 180,E1 26626.606,E2 26626.606} C_VEL
LIN {X 0,Y 552.807,Z 500.166,A -85,B 0,C 180,E1 26624.983,E2 26624.983} C_VEL
LIN {X 0,Y 553.119,Z 487.937,A -85,B 0,C 180,E1 26623.716,E2 26623.716} C_VEL
LIN {X 0,Y 553.53,Z 473.575,A -85,B 0,C 180,E1 26622.443,E2 26622.443} C_VEL
LIN {X 0,Y 553.936,Z 458.008,A -85,B 0,C 180,E1 26621.314,E2 26621.314} C_VEL
LIN {X 0,Y 554.367,Z 441.837,A -85,B 0,C 180,E1 26620.339,E2 26620.339} C_VEL
LIN {X 0,Y 554.68,Z 425.964,A -85,B 0,C 180,E1 26619.586,E2 26619.586} C_VEL
LIN {X 0,Y 555.012,Z 407.702,A -85,B 0,C 180,E1 26618.912,E2 26618.912} C_VEL
LIN {X 0,Y 555.237,Z 389.419,A -85,B 0,C 180,E1 26618.44,E2 26618.44} C_VEL
LIN {X 0,Y 555.391,Z 365.319,A -85,B 0,C 180,E1 26618.065,E2 26618.065} C_VEL
LIN {X 0,Y 556.116,Z 182.899,A -85,B 0,C 180,E1 26615.594,E2 26615.594} C_VEL
LIN {X 0,Y 555.19,Z 177.501,A -85,B 0,C 180,E1 26615.474,E2 26615.474} C_VEL
LIN {X 0,Y 555.46,Z 143.156,A -85,B 0,C 180,E1 26612.851,E2 26612.851} C_VEL
LIN {X 0,Y 555.352,Z 111.338,A -85,B 0,C 180,E1 26610.501,E2 26610.501} C_VEL
LIN {X 0,Y 552.345,Z 100.686,A -85,B 0,C 180,E1 26609.576,E2 26609.576} C_VEL
LIN {X 0,Y 552.298,Z 100.686,A -85,B 0,C 180,E1 26606.36,E2 26606.36} C_VEL
LIN {X 0,Y 552.307,Z 100.688,A -85,B 0,C 180,E1 26602.974,E2 26602.974} C_VEL
LIN {X 0,Y 552.345,Z 100.686,A -85,B 0,C 180,E1 26599.65,E2 26599.65} C_VEL
LIN {X 0,Y 552.282,Z 100.688,A -85,B 0,C 180,E1 26596.389,E2 26596.389} C_VEL
LIN {X 0,Y 552.273,Z 100.689,A -85,B 0,C 180,E1 26592.995,E2 26592.995} C_VEL
LIN {X 0,Y 552.33,Z 100.688,A -85,B 0,C 180,E1 26589.704,E2 26589.704} C_VEL
LIN {X 0,Y 552.283,Z 100.691,A -85,B 0,C 180,E1 26586.504,E2 26586.504} C_VEL
LIN {X 0,Y 552.286,Z 100.757,A -85,B 0,C 180,E1 26584.961,E2 26584.961} C_VEL
LIN {X 0,Y 558.377,Z 116.941,A -85,B 0,C 180,E1 26583.472,E2 26583.472} C_VEL
LIN {X 0,Y 557.367,Z 163.122,A -85,B 0,C 180,E1 26580.45,E2 26580.45} C_VEL
LIN {X 0,Y 558.771,Z 173.104,A -85,B 0,C 180,E1 26580.219,E2 26580.219} C_VEL
LIN {X 0,Y 557.344,Z 412.49,A -85,B 0,C 180,E1 26576.863,E2 26576.863} C_VEL
LIN {X 0,Y 557.101,Z 433.492,A -85,B 0,C 180,E1 26576.488,E2 26576.488} C_VEL
LIN {X 0,Y 556.688,Z 454.216,A -85,B 0,C 180,E1 26575.925,E2 26575.925} C_VEL
LIN {X 0,Y 556.206,Z 474.695,A -85,B 0,C 180,E1 26575.16,E2 26575.16} C_VEL
LIN {X 0,Y 555.685,Z 493.262,A -85,B 0,C 180,E1 26574.277,E2 26574.277} C_VEL
LIN {X 0,Y 555.099,Z 512.067,A -85,B 0,C 180,E1 26573.177,E2 26573.177} C_VEL
LIN {X 0,Y 554.479,Z 530.551,A -85,B 0,C 180,E1 26571.862,E2 26571.862} C_VEL
LIN {X 0,Y 553.927,Z 546.87,A -85,B 0,C 180,E1 26570.477,E2 26570.477} C_VEL
LIN {X 0,Y 553.412,Z 562.45,A -85,B 0,C 180,E1 26568.924,E2 26568.924} C_VEL
LIN {X 0,Y 552.97,Z 576.749,A -85,B 0,C 180,E1 26567.25,E2 26567.25} C_VEL
LIN {X 0,Y 552.608,Z 589.977,A -85,B 0,C 180,E1 26565.425,E2 26565.425} C_VEL
LIN {X 0,Y 552.334,Z 601.351,A -85,B 0,C 180,E1 26563.567,E2 26563.567} C_VEL
LIN {X 0,Y 552.143,Z 611.52,A -85,B 0,C 180,E1 26561.571,E2 26561.571} C_VEL
LIN {X 0,Y 552.019,Z 620.086,A -85,B 0,C 180,E1 26559.488,E2 26559.488} C_VEL
LIN {X 0,Y 551.951,Z 626.503,A -85,B 0,C 180,E1 26557.495,E2 26557.495} C_VEL
LIN {X 0,Y 551.917,Z 631.555,A -85,B 0,C 180,E1 26555.406,E2 26555.406} C_VEL
LIN {X 0,Y 551.906,Z 634.941,A -85,B 0,C 180,E1 26553.324,E2 26553.324} C_VEL
LIN {X 0,Y 551.909,Z 636.759,A -85,B 0,C 180,E1 26551.143,E2 26551.143} C_VEL
LIN {X 0,Y 551.913,Z 636.783,A -85,B 0,C 180,E1 26548.963,E2 26548.963} C_VEL
LIN {X 0,Y 551.913,Z 635.169,A -85,B 0,C 180,E1 26546.885,E2 26546.885} C_VEL
LIN {X 0,Y 551.917,Z 631.762,A -85,B 0,C 180,E1 26544.699,E2 26544.699} C_VEL
LIN {X 0,Y 551.95,Z 626.811,A -85,B 0,C 180,E1 26542.611,E2 26542.611} C_VEL
LIN {X 0,Y 552.018,Z 620.492,A -85,B 0,C 180,E1 26540.619,E2 26540.619} C_VEL
LIN {X 0,Y 552.14,Z 611.877,A -85,B 0,C 180,E1 26538.511,E2 26538.511} C_VEL
LIN {X 0,Y 552.317,Z 602.268,A -85,B 0,C 180,E1 26536.603,E2 26536.603} C_VEL
LIN {X 0,Y 552.592,Z 590.588,A -85,B 0,C 180,E1 26534.667,E2 26534.667} C_VEL
LIN {X 0,Y 552.944,Z 577.605,A -85,B 0,C 180,E1 26532.859,E2 26532.859} C_VEL
LIN {X 0,Y 553.397,Z 562.968,A -85,B 0,C 180,E1 26531.131,E2 26531.131} C_VEL
LIN {X 0,Y 553.893,Z 547.857,A -85,B 0,C 180,E1 26529.612,E2 26529.612} C_VEL
LIN {X 0,Y 554.454,Z 531.286,A -85,B 0,C 180,E1 26528.194,E2 26528.194} C_VEL
LIN {X 0,Y 555.069,Z 512.904,A -85,B 0,C 180,E1 26526.879,E2 26526.879} C_VEL
LIN {X 0,Y 555.649,Z 494.286,A -85,B 0,C 180,E1 26525.779,E2 26525.779} C_VEL
LIN {X 0,Y 556.165,Z 476.007,A -85,B 0,C 180,E1 26524.896,E2 26524.896} C_VEL
LIN {X 0,Y 556.664,Z 455.673,A -85,B 0,C 180,E1 26524.122,E2 26524.122} C_VEL
LIN {X 0,Y 557.084,Z 435.51,A -85,B 0,C 180,E1 26523.556,E2 26523.556} C_VEL
LIN {X 0,Y 557.333,Z 414.501,A -85,B 0,C 180,E1 26523.165,E2 26523.165} C_VEL
LIN {X 0,Y 558.749,Z 176.061,A -85,B 0,C 180,E1 26519.822,E2 26519.822} C_VEL
LIN {X 0,Y 558.503,Z 170.019,A -85,B 0,C 180,E1 26519.72,E2 26519.72} C_VEL
LIN {X 0,Y 557.331,Z 162.864,A -85,B 0,C 180,E1 26519.544,E2 26519.544} C_VEL
LIN {X 0,Y 558.389,Z 116.509,A -85,B 0,C 180,E1 26516.5,E2 26516.5} C_VEL
LIN {X 0,Y 552.285,Z 100.691,A -85,B 0,C 180,E1 26515.013,E2 26515.013} C_VEL
LIN {X 0,Y 552.321,Z 100.688,A -85,B 0,C 180,E1 26511.749,E2 26511.749} C_VEL
LIN {X 0,Y 552.301,Z 100.684,A -85,B 0,C 180,E1 26508.642,E2 26508.642} C_VEL
LIN {X 0,Y 552.288,Z 100.687,A -85,B 0,C 180,E1 26505.356,E2 26505.356} C_VEL
LIN {X 0,Y 552.344,Z 100.684,A -85,B 0,C 180,E1 26502.083,E2 26502.083} C_VEL
LIN {X 0,Y 552.286,Z 100.672,A -85,B 0,C 180,E1 26498.881,E2 26498.881} C_VEL
LIN {X 0,Y 552.284,Z 100.687,A -85,B 0,C 180,E1 26495.446,E2 26495.446} C_VEL
LIN {X 0,Y 552.338,Z 100.68,A -85,B 0,C 180,E1 26492.277,E2 26492.277} C_VEL
LIN {X 0,Y 552.279,Z 100.683,A -85,B 0,C 180,E1 26489.144,E2 26489.144} C_VEL
LIN {X 0,Y 552.309,Z 100.686,A -85,B 0,C 180,E1 26485.867,E2 26485.867} C_VEL
LIN {X 0,Y 552.306,Z 100.682,A -85,B 0,C 180,E1 26482.681,E2 26482.681} C_VEL
LIN {X 0,Y 552.277,Z 100.681,A -85,B 0,C 180,E1 26479.401,E2 26479.401} C_VEL
LIN {X 0,Y 552.335,Z 100.688,A -85,B 0,C 180,E1 26476.187,E2 26476.187} C_VEL
LIN {X 0,Y 552.279,Z 100.679,A -85,B 0,C 180,E1 26473.079,E2 26473.079} C_VEL
LIN {X 0,Y 552.282,Z 100.687,A -85,B 0,C 180,E1 26469.693,E2 26469.693} C_VEL
LIN {X 0,Y 552.342,Z 100.677,A -85,B 0,C 180,E1 26466.444,E2 26466.444} C_VEL
LIN {X 0,Y 552.275,Z 100.686,A -85,B 0,C 180,E1 26463.217,E2 26463.217} C_VEL
LIN {X 0,Y 552.289,Z 100.685,A -85,B 0,C 180,E1 26459.896,E2 26459.896} C_VEL
LIN {X 0,Y 552.308,Z 100.686,A -85,B 0,C 180,E1 26456.783,E2 26456.783} C_VEL
LIN {X 0,Y 552.269,Z 100.684,A -85,B 0,C 180,E1 26453.555,E2 26453.555} C_VEL
LIN {X 0,Y 552.331,Z 100.685,A -85,B 0,C 180,E1 26450.413,E2 26450.413} C_VEL
LIN {X 0,Y 552.275,Z 100.683,A -85,B 0,C 180,E1 26447.239,E2 26447.239} C_VEL
LIN {X 0,Y 552.271,Z 100.685,A -85,B 0,C 180,E1 26443.811,E2 26443.811} C_VEL
LIN {X 0,Y 552.332,Z 100.684,A -85,B 0,C 180,E1 26440.583,E2 26440.583} C_VEL
LIN {X 0,Y 552.268,Z 100.683,A -85,B 0,C 180,E1 26437.416,E2 26437.416} C_VEL
LIN {X 0,Y 552.277,Z 100.687,A -85,B 0,C 180,E1 26434.016,E2 26434.016} C_VEL
LIN {X 0,Y 552.327,Z 100.686,A -85,B 0,C 180,E1 26432.726,E2 26432.726} C_VEL
LIN {X 0,Y 551.335,Z 100.8,A -85,B 0,C 180,E1 26431.926,E2 26431.926} C_VEL
LIN {X 0,Y 544.847,Z 101.612,A -85,B 0,C 180,E1 26429.684,E2 26429.684} C_VEL
LIN {X 0,Y 544.35,Z 101.676,A -85,B 0,C 180,E1 26429.099,E2 26429.099} C_VEL
LIN {X 0,Y 544.324,Z 101.676,A -85,B 0,C 180,E1 26425.749,E2 26425.749} C_VEL
LIN {X 0,Y 544.375,Z 101.674,A -85,B 0,C 180,E1 26422.508,E2 26422.508} C_VEL
LIN {X 0,Y 544.334,Z 101.676,A -85,B 0,C 180,E1 26419.341,E2 26419.341} C_VEL
LIN {X 0,Y 544.328,Z 101.674,A -85,B 0,C 180,E1 26416.025,E2 26416.025} C_VEL
LIN {X 0,Y 544.388,Z 101.674,A -85,B 0,C 180,E1 26412.809,E2 26412.809} C_VEL
LIN {X 0,Y 544.325,Z 101.677,A -85,B 0,C 180,E1 26409.597,E2 26409.597} C_VEL
LIN {X 0,Y 544.34,Z 101.677,A -85,B 0,C 180,E1 26406.257,E2 26406.257} C_VEL
LIN {X 0,Y 544.373,Z 101.679,A -85,B 0,C 180,E1 26403.058,E2 26403.058} C_VEL
LIN {X 0,Y 544.352,Z 101.833,A -85,B 0,C 180,E1 26401.565,E2 26401.565} C_VEL
LIN {X 0,Y 549.532,Z 117.425,A -85,B 0,C 180,E1 26399.842,E2 26399.842} C_VEL
LIN {X 0,Y 548.409,Z 156.183,A -85,B 0,C 180,E1 26396.589,E2 26396.589} C_VEL
LIN {X 0,Y 547.974,Z 175.266,A -85,B 0,C 180,E1 26395.038,E2 26395.038} C_VEL
LIN {X 0,Y 549.663,Z 185.95,A -85,B 0,C 180,E1 26394.796,E2 26394.796} C_VEL
LIN {X 0,Y 548.545,Z 383.629,A -85,B 0,C 180,E1 26392.059,E2 26392.059} C_VEL
LIN {X 0,Y 548.221,Z 402.538,A -85,B 0,C 180,E1 26391.61,E2 26391.61} C_VEL
LIN {X 0,Y 547.768,Z 421.037,A -85,B 0,C 180,E1 26390.962,E2 26390.962} C_VEL
LIN {X 0,Y 547.221,Z 438.307,A -85,B 0,C 180,E1 26390.154,E2 26390.154} C_VEL
LIN {X 0,Y 546.635,Z 454.945,A -85,B 0,C 180,E1 26389.166,E2 26389.166} C_VEL
LIN {X 0,Y 546.011,Z 471.202,A -85,B 0,C 180,E1 26387.972,E2 26387.972} C_VEL
LIN {X 0,Y 545.446,Z 485.785,A -85,B 0,C 180,E1 26386.671,E2 26386.671} C_VEL
LIN {X 0,Y 544.921,Z 501.493,A -85,B 0,C 180,E1 26384.993,E2 26384.993} C_VEL
LIN {X 0,Y 544.572,Z 514.138,A -85,B 0,C 180,E1 26383.375,E2 26383.375} C_VEL
LIN {X 0,Y 544.303,Z 525.237,A -85,B 0,C 180,E1 26381.657,E2 26381.657} C_VEL
LIN {X 0,Y 544.121,Z 534.808,A -85,B 0,C 180,E1 26379.839,E2 26379.839} C_VEL
LIN {X 0,Y 544.009,Z 542.414,A -85,B 0,C 180,E1 26378.029,E2 26378.029} C_VEL
LIN {X 0,Y 543.946,Z 548.591,A -85,B 0,C 180,E1 26376.119,E2 26376.119} C_VEL
LIN {X 0,Y 543.921,Z 552.996,A -85,B 0,C 180,E1 26374.216,E2 26374.216} C_VEL
LIN {X 0,Y 543.915,Z 555.858,A -85,B 0,C 180,E1 26372.212,E2 26372.212} C_VEL
LIN {X 0,Y 543.911,Z 556.952,A -85,B 0,C 180,E1 26370.21,E2 26370.21} C_VEL
LIN {X 0,Y 543.914,Z 556.307,A -85,B 0,C 180,E1 26368.209,E2 26368.209} C_VEL
LIN {X 0,Y 543.912,Z 554.068,A -85,B 0,C 180,E1 26366.31,E2 26366.31} C_VEL
LIN {X 0,Y 543.934,Z 550.201,A -85,B 0,C 180,E1 26364.408,E2 26364.408} C_VEL
LIN {X 0,Y 543.977,Z 544.612,A -85,B 0,C 180,E1 26362.501,E2 26362.501} C_VEL
LIN {X 0,Y 544.078,Z 537.158,A -85,B 0,C 180,E1 26360.586,E2 26360.586} C_VEL
LIN {X 0,Y 544.242,Z 528.18,A -85,B 0,C 180,E1 26358.77,E2 26358.77} C_VEL
LIN {X 0,Y 544.478,Z 517.737,A -85,B 0,C 180,E1 26357.053,E2 26357.053} C_VEL
LIN {X 0,Y 544.799,Z 505.85,A -85,B 0,C 180,E1 26355.437,E2 26355.437} C_VEL
LIN {X 0,Y 545.22,Z 491.987,A -85,B 0,C 180,E1 26353.869,E2 26353.869} C_VEL
LIN {X 0,Y 545.764,Z 477.677,A -85,B 0,C 180,E1 26352.484,E2 26352.484} C_VEL
LIN {X 0,Y 546.385,Z 461.697,A -85,B 0,C 180,E1 26351.211,E2 26351.211} C_VEL
LIN {X 0,Y 546.965,Z 445.852,A -85,B 0,C 180,E1 26350.178,E2 26350.178} C_VEL
LIN {X 0,Y 547.522,Z 429.252,A -85,B 0,C 180,E1 26349.306,E2 26349.306} C_VEL
LIN {X 0,Y 548.024,Z 411.01,A -85,B 0,C 180,E1 26348.571,E2 26348.571} C_VEL
LIN {X 0,Y 548.408,Z 392.535,A -85,B 0,C 180,E1 26348.038,E2 26348.038} C_VEL
LIN {X 0,Y 548.636,Z 372.859,A -85,B 0,C 180,E1 26347.681,E2 26347.681} C_VEL
LIN {X 0,Y 549.585,Z 184.099,A -85,B 0,C 180,E1 26345.088,E2 26345.088} C_VEL
LIN {X 0,Y 547.916,Z 174.572,A -85,B 0,C 180,E1 26344.837,E2 26344.837} C_VEL
LIN {X 0,Y 549.011,Z 135.057,A -85,B 0,C 180,E1 26341.559,E2 26341.559} C_VEL
LIN {X 0,Y 549.488,Z 116.837,A -85,B 0,C 180,E1 26340.014,E2 26340.014} C_VEL
LIN {X 0,Y 544.333,Z 101.682,A -85,B 0,C 180,E1 26338.308,E2 26338.308} C_VEL
LIN {X 0,Y 544.385,Z 101.675,A -85,B 0,C 180,E1 26335.037,E2 26335.037} C_VEL
LIN {X 0,Y 544.384,Z 101.665,A -85,B 0,C 180,E1 26331.759,E2 26331.759} C_VEL
LIN {X 0,Y 544.366,Z 101.675,A -85,B 0,C 180,E1 26328.466,E2 26328.466} C_VEL
LIN {X 0,Y 544.397,Z 101.67,A -85,B 0,C 180,E1 26325.148,E2 26325.148} C_VEL
LIN {X 0,Y 544.397,Z 101.673,A -85,B 0,C 180,E1 26321.782,E2 26321.782} C_VEL
LIN {X 0,Y 544.401,Z 101.675,A -85,B 0,C 180,E1 26318.349,E2 26318.349} C_VEL
LIN {X 0,Y 544.398,Z 101.673,A -85,B 0,C 180,E1 26314.962,E2 26314.962} C_VEL
LIN {X 0,Y 544.389,Z 101.674,A -85,B 0,C 180,E1 26311.546,E2 26311.546} C_VEL
LIN {X 0,Y 544.426,Z 101.835,A -85,B 0,C 180,E1 26311.035,E2 26311.035} C_VEL
LIN {X 0,Y 548.58,Z 115.217,A -85,B 0,C 180,E1 26309.72,E2 26309.72} C_VEL
LIN {X 0,Y 547.987,Z 155.819,A -85,B 0,C 180,E1 26306.495,E2 26306.495} C_VEL
LIN {X 0,Y 547.699,Z 177.23,A -85,B 0,C 180,E1 26304.818,E2 26304.818} C_VEL
LIN {X 0,Y 548.88,Z 186.098,A -85,B 0,C 180,E1 26304.629,E2 26304.629} C_VEL
LIN {X 0,Y 547.784,Z 385.341,A -85,B 0,C 180,E1 26301.844,E2 26301.844} C_VEL
LIN {X 0,Y 547.531,Z 404.118,A -85,B 0,C 180,E1 26301.39,E2 26301.39} C_VEL
LIN {X 0,Y 547.195,Z 422.223,A -85,B 0,C 180,E1 26300.762,E2 26300.762} C_VEL
LIN {X 0,Y 546.758,Z 440.277,A -85,B 0,C 180,E1 26299.922,E2 26299.922} C_VEL
LIN {X 0,Y 546.303,Z 456.594,A -85,B 0,C 180,E1 26298.958,E2 26298.958} C_VEL
LIN {X 0,Y 545.834,Z 472.452,A -85,B 0,C 180,E1 26297.813,E2 26297.813} C_VEL
LIN {X 0,Y 545.364,Z 486.575,A -85,B 0,C 180,E1 26296.564,E2 26296.564} C_VEL
LIN {X 0,Y 544.974,Z 499.806,A -85,B 0,C 180,E1 26295.192,E2 26295.192} C_VEL
LIN {X 0,Y 544.625,Z 511.757,A -85,B 0,C 180,E1 26293.7,E2 26293.7} C_VEL
LIN {X 0,Y 544.383,Z 521.424,A -85,B 0,C 180,E1 26292.28,E2 26292.28} C_VEL
LIN {X 0,Y 544.19,Z 531.166,A -85,B 0,C 180,E1 26290.586,E2 26290.586} C_VEL
LIN {X 0,Y 544.042,Z 539.463,A -85,B 0,C 180,E1 26288.774,E2 26288.774} C_VEL
LIN {X 0,Y 543.967,Z 546.084,A -85,B 0,C 180,E1 26286.968,E2 26286.968} C_VEL
LIN {X 0,Y 543.922,Z 551.229,A -85,B 0,C 180,E1 26285.062,E2 26285.062} C_VEL
LIN {X 0,Y 543.912,Z 554.545,A -85,B 0,C 180,E1 26283.267,E2 26283.267} C_VEL
LIN {X 0,Y 543.909,Z 556.617,A -85,B 0,C 180,E1 26281.264,E2 26281.264} C_VEL
LIN {X 0,Y 543.915,Z 556.851,A -85,B 0,C 180,E1 26279.368,E2 26279.368} C_VEL
LIN {X 0,Y 543.913,Z 555.643,A -85,B 0,C 180,E1 26277.472,E2 26277.472} C_VEL
LIN {X 0,Y 543.922,Z 552.531,A -85,B 0,C 180,E1 26275.467,E2 26275.467} C_VEL
LIN {X 0,Y 543.948,Z 548.236,A -85,B 0,C 180,E1 26273.668,E2 26273.668} C_VEL
LIN {X 0,Y 544.013,Z 541.534,A -85,B 0,C 180,E1 26271.652,E2 26271.652} C_VEL
LIN {X 0,Y 544.126,Z 534.184,A -85,B 0,C 180,E1 26269.947,E2 26269.947} C_VEL
LIN {X 0,Y 544.325,Z 524.518,A -85,B 0,C 180,E1 26268.128,E2 26268.128} C_VEL
LIN {X 0,Y 544.549,Z 514.721,A -85,B 0,C 180,E1 26266.624,E2 26266.624} C_VEL
LIN {X 0,Y 544.877,Z 503.181,A -85,B 0,C 180,E1 26265.114,E2 26265.114} C_VEL
LIN {X 0,Y 545.274,Z 489.724,A -85,B 0,C 180,E1 26263.652,E2 26263.652} C_VEL
LIN {X 0,Y 545.678,Z 477.013,A -85,B 0,C 180,E1 26262.48,E2 26262.48} C_VEL
LIN {X 0,Y 546.166,Z 461.126,A -85,B 0,C 180,E1 26261.26,E2 26261.26} C_VEL
LIN {X 0,Y 546.597,Z 445.373,A -85,B 0,C 180,E1 26260.276,E2 26260.276} C_VEL
LIN {X 0,Y 547.005,Z 427.51,A -85,B 0,C 180,E1 26259.393,E2 26259.393} C_VEL
LIN {X 0,Y 547.353,Z 409.124,A -85,B 0,C 180,E1 26258.702,E2 26258.702} C_VEL
LIN {X 0,Y 547.598,Z 390.537,A -85,B 0,C 180,E1 26258.211,E2 26258.211} C_VEL
LIN {X 0,Y 547.747,Z 368.592,A -85,B 0,C 180,E1 26257.857,E2 26257.857} C_VEL
LIN {X 0,Y 548.692,Z 195.671,A -85,B 0,C 180,E1 26255.464,E2 26255.464} C_VEL
LIN {X 0,Y 548.555,Z 183.095,A -85,B 0,C 180,E1 26255.269,E2 26255.269} C_VEL
LIN {X 0,Y 547.779,Z 178.281,A -85,B 0,C 180,E1 26255.148,E2 26255.148} C_VEL
LIN {X 0,Y 548.019,Z 142.999,A -85,B 0,C 180,E1 26252.463,E2 26252.463} C_VEL
LIN {X 0,Y 547.892,Z 113.708,A -85,B 0,C 180,E1 26250.304,E2 26250.304} C_VEL
LIN {X 0,Y 544.407,Z 101.675,A -85,B 0,C 180,E1 26249.265,E2 26249.265} C_VEL
LIN {X 0,Y 544.382,Z 101.674,A -85,B 0,C 180,E1 26245.93,E2 26245.93} C_VEL
LIN {X 0,Y 544.352,Z 101.676,A -85,B 0,C 180,E1 26242.557,E2 26242.557} C_VEL
LIN {X 0,Y 544.383,Z 101.678,A -85,B 0,C 180,E1 26239.306,E2 26239.306} C_VEL
LIN {X 0,Y 544.369,Z 101.676,A -85,B 0,C 180,E1 26236.03,E2 26236.03} C_VEL
LIN {X 0,Y 544.329,Z 101.678,A -85,B 0,C 180,E1 26232.816,E2 26232.816} C_VEL
LIN {X 0,Y 544.368,Z 101.679,A -85,B 0,C 180,E1 26229.518,E2 26229.518} C_VEL
LIN {X 0,Y 544.352,Z 101.681,A -85,B 0,C 180,E1 26226.391,E2 26226.391} C_VEL
LIN {X 0,Y 544.369,Z 101.73,A -85,B 0,C 180,E1 26225.435,E2 26225.435} C_VEL
LIN {X 0,Y 551.252,Z 119.541,A -85,B 0,C 180,E1 26223.75,E2 26223.75} C_VEL
LIN {X 0,Y 550.306,Z 163.458,A -85,B 0,C 180,E1 26220.878,E2 26220.878} C_VEL
LIN {X 0,Y 551.849,Z 174.406,A -85,B 0,C 180,E1 26220.62,E2 26220.62} C_VEL
LIN {X 0,Y 550.2,Z 413.889,A -85,B 0,C 180,E1 26217.221,E2 26217.221} C_VEL
LIN {X 0,Y 549.913,Z 434.79,A -85,B 0,C 180,E1 26216.832,E2 26216.832} C_VEL
LIN {X 0,Y 549.44,Z 455.082,A -85,B 0,C 180,E1 26216.263,E2 26216.263} C_VEL
LIN {X 0,Y 548.907,Z 474.692,A -85,B 0,C 180,E1 26215.519,E2 26215.519} C_VEL
LIN {X 0,Y 548.302,Z 493.259,A -85,B 0,C 180,E1 26214.626,E2 26214.626} C_VEL
LIN {X 0,Y 547.63,Z 512.066,A -85,B 0,C 180,E1 26213.512,E2 26213.512} C_VEL
LIN {X 0,Y 546.945,Z 529.827,A -85,B 0,C 180,E1 26212.236,E2 26212.236} C_VEL
LIN {X 0,Y 546.282,Z 546.638,A -85,B 0,C 180,E1 26210.799,E2 26210.799} C_VEL
LIN {X 0,Y 545.689,Z 561.943,A -85,B 0,C 180,E1 26209.258,E2 26209.258} C_VEL
LIN {X 0,Y 545.154,Z 576.796,A -85,B 0,C 180,E1 26207.499,E2 26207.499} C_VEL
LIN {X 0,Y 544.732,Z 589.978,A -85,B 0,C 180,E1 26205.654,E2 26205.654} C_VEL
LIN {X 0,Y 544.4,Z 601.685,A -85,B 0,C 180,E1 26203.706,E2 26203.706} C_VEL
LIN {X 0,Y 544.183,Z 611.408,A -85,B 0,C 180,E1 26201.768,E2 26201.768} C_VEL
LIN {X 0,Y 544.039,Z 619.68,A -85,B 0,C 180,E1 26199.735,E2 26199.735} C_VEL
LIN {X 0,Y 543.968,Z 626.2,A -85,B 0,C 180,E1 26197.712,E2 26197.712} C_VEL
LIN {X 0,Y 543.924,Z 631.347,A -85,B 0,C 180,E1 26195.592,E2 26195.592} C_VEL
LIN {X 0,Y 543.907,Z 634.827,A -85,B 0,C 180,E1 26193.479,E2 26193.479} C_VEL
LIN {X 0,Y 543.905,Z 636.707,A -85,B 0,C 180,E1 26191.265,E2 26191.265} C_VEL
LIN {X 0,Y 543.911,Z 636.828,A -85,B 0,C 180,E1 26189.158,E2 26189.158} C_VEL
LIN {X 0,Y 543.914,Z 635.282,A -85,B 0,C 180,E1 26186.945,E2 26186.945} C_VEL
LIN {X 0,Y 543.919,Z 631.967,A -85,B 0,C 180,E1 26184.727,E2 26184.727} C_VEL
LIN {X 0,Y 543.955,Z 627.114,A -85,B 0,C 180,E1 26182.608,E2 26182.608} C_VEL
LIN {X 0,Y 544.036,Z 620.492,A -85,B 0,C 180,E1 26180.48,E2 26180.48} C_VEL
LIN {X 0,Y 544.174,Z 611.878,A -85,B 0,C 180,E1 26178.34,E2 26178.34} C_VEL
LIN {X 0,Y 544.387,Z 602.27,A -85,B 0,C 180,E1 26176.404,E2 26176.404} C_VEL
LIN {X 0,Y 544.711,Z 590.693,A -85,B 0,C 180,E1 26174.456,E2 26174.456} C_VEL
LIN {X 0,Y 545.129,Z 577.604,A -85,B 0,C 180,E1 26172.605,E2 26172.605} C_VEL
LIN {X 0,Y 545.654,Z 562.968,A -85,B 0,C 180,E1 26170.853,E2 26170.853} C_VEL
LIN {X 0,Y 546.252,Z 547.514,A -85,B 0,C 180,E1 26169.282,E2 26169.282} C_VEL
LIN {X 0,Y 546.907,Z 530.841,A -85,B 0,C 180,E1 26167.841,E2 26167.841} C_VEL
LIN {X 0,Y 547.59,Z 512.901,A -85,B 0,C 180,E1 26166.544,E2 26166.544} C_VEL
LIN {X 0,Y 548.222,Z 495.388,A -85,B 0,C 180,E1 26165.492,E2 26165.492} C_VEL
LIN {X 0,Y 548.862,Z 476.004,A -85,B 0,C 180,E1 26164.538,E2 26164.538} C_VEL
LIN {X 0,Y 549.424,Z 455.813,A -85,B 0,C 180,E1 26163.76,E2 26163.76} C_VEL
LIN {X 0,Y 549.905,Z 435.673,A -85,B 0,C 180,E1 26163.187,E2 26163.187} C_VEL
LIN {X 0,Y 550.196,Z 414.501,A -85,B 0,C 180,E1 26162.788,E2 26162.788} C_VEL
LIN {X 0,Y 551.839,Z 175.552,A -85,B 0,C 180,E1 26159.397,E2 26159.397} C_VEL
LIN {X 0,Y 551.469,Z 170.56,A -85,B 0,C 180,E1 26159.3,E2 26159.3} C_VEL
LIN {X 0,Y 550.228,Z 162.496,A -85,B 0,C 180,E1 26159.083,E2 26159.083} C_VEL
LIN {X 0,Y 551.259,Z 119.425,A -85,B 0,C 180,E1 26156.241,E2 26156.241} C_VEL
LIN {X 0,Y 544.366,Z 101.679,A -85,B 0,C 180,E1 26154.557,E2 26154.557} C_VEL
LIN {X 0,Y 544.346,Z 101.675,A -85,B 0,C 180,E1 26151.22,E2 26151.22} C_VEL
LIN {X 0,Y 544.401,Z 101.671,A -85,B 0,C 180,E1 26148.047,E2 26148.047} C_VEL
LIN {X 0,Y 544.35,Z 101.675,A -85,B 0,C 180,E1 26144.848,E2 26144.848} C_VEL
LIN {X 0,Y 544.349,Z 101.675,A -85,B 0,C 180,E1 26141.395,E2 26141.395} C_VEL
LIN {X 0,Y 544.401,Z 101.654,A -85,B 0,C 180,E1 26138.105,E2 26138.105} C_VEL
LIN {X 0,Y 544.352,Z 101.674,A -85,B 0,C 180,E1 26134.812,E2 26134.812} C_VEL
LIN {X 0,Y 544.345,Z 101.676,A -85,B 0,C 180,E1 26131.443,E2 26131.443} C_VEL
LIN {X 0,Y 544.406,Z 101.669,A -85,B 0,C 180,E1 26128.164,E2 26128.164} C_VEL
LIN {X 0,Y 544.352,Z 101.673,A -85,B 0,C 180,E1 26124.858,E2 26124.858} C_VEL
LIN {X 0,Y 544.344,Z 101.676,A -85,B 0,C 180,E1 26121.553,E2 26121.553} C_VEL
LIN {X 0,Y 544.399,Z 101.668,A -85,B 0,C 180,E1 26118.283,E2 26118.283} C_VEL
LIN {X 0,Y 544.345,Z 101.674,A -85,B 0,C 180,E1 26115.01,E2 26115.01} C_VEL
LIN {X 0,Y 544.344,Z 101.675,A -85,B 0,C 180,E1 26111.657,E2 26111.657} C_VEL
LIN {X 0,Y 544.398,Z 101.673,A -85,B 0,C 180,E1 26108.449,E2 26108.449} C_VEL
LIN {X 0,Y 544.335,Z 101.674,A -85,B 0,C 180,E1 26105.269,E2 26105.269} C_VEL
LIN {X 0,Y 544.351,Z 101.669,A -85,B 0,C 180,E1 26101.894,E2 26101.894} C_VEL
LIN {X 0,Y 544.372,Z 101.672,A -85,B 0,C 180,E1 26098.737,E2 26098.737} C_VEL
LIN {X 0,Y 544.329,Z 101.671,A -85,B 0,C 180,E1 26095.47,E2 26095.47} C_VEL
LIN {X 0,Y 544.371,Z 101.677,A -85,B 0,C 180,E1 26092.188,E2 26092.188} C_VEL
LIN {X 0,Y 544.352,Z 101.672,A -85,B 0,C 180,E1 26088.987,E2 26088.987} C_VEL
LIN {X 0,Y 544.33,Z 101.676,A -85,B 0,C 180,E1 26085.642,E2 26085.642} C_VEL
LIN {X 0,Y 544.385,Z 101.669,A -85,B 0,C 180,E1 26082.405,E2 26082.405} C_VEL
LIN {X 0,Y 544.339,Z 101.676,A -85,B 0,C 180,E1 26079.217,E2 26079.217} C_VEL
LIN {X 0,Y 544.329,Z 101.674,A -85,B 0,C 180,E1 26075.819,E2 26075.819} C_VEL
LIN {X 0,Y 544.389,Z 101.67,A -85,B 0,C 180,E1 26072.548,E2 26072.548} C_VEL
LIN {X 0,Y 544.335,Z 101.676,A -85,B 0,C 180,E1 26069.293,E2 26069.293} C_VEL
LIN {X 0,Y 544.35,Z 101.676,A -85,B 0,C 180,E1 26069.099,E2 26069.099} C_VEL
LIN {X 0,Y 543.401,Z 101.799,A -85,B 0,C 180,E1 26068.288,E2 26068.288} C_VEL
LIN {X 0,Y 536.915,Z 102.601,A -85,B 0,C 180,E1 26066.01,E2 26066.01} C_VEL
LIN {X 0,Y 536.39,Z 102.665,A -85,B 0,C 180,E1 26065.417,E2 26065.417} C_VEL
LIN {X 0,Y 536.393,Z 102.665,A -85,B 0,C 180,E1 26062.038,E2 26062.038} C_VEL
LIN {X 0,Y 536.446,Z 102.661,A -85,B 0,C 180,E1 26058.849,E2 26058.849} C_VEL
LIN {X 0,Y 536.385,Z 102.663,A -85,B 0,C 180,E1 26055.555,E2 26055.555} C_VEL
LIN {X 0,Y 536.392,Z 102.668,A -85,B 0,C 180,E1 26052.107,E2 26052.107} C_VEL
LIN {X 0,Y 536.455,Z 102.667,A -85,B 0,C 180,E1 26048.823,E2 26048.823} C_VEL
LIN {X 0,Y 536.39,Z 102.667,A -85,B 0,C 180,E1 26045.561,E2 26045.561} C_VEL
LIN {X 0,Y 536.398,Z 102.726,A -85,B 0,C 180,E1 26042.049,E2 26042.049} C_VEL
LIN {X 0,Y 542.311,Z 119.934,A -85,B 0,C 180,E1 26040.097,E2 26040.097} C_VEL
LIN {X 0,Y 541.016,Z 159.442,A -85,B 0,C 180,E1 26036.744,E2 26036.744} C_VEL
LIN {X 0,Y 540.649,Z 175.31,A -85,B 0,C 180,E1 26035.45,E2 26035.45} C_VEL
LIN {X 0,Y 542.579,Z 186.939,A -85,B 0,C 180,E1 26035.177,E2 26035.177} C_VEL
LIN {X 0,Y 541.424,Z 383.921,A -85,B 0,C 180,E1 26032.441,E2 26032.441} C_VEL
LIN {X 0,Y 541.077,Z 402.536,A -85,B 0,C 180,E1 26031.999,E2 26031.999} C_VEL
LIN {X 0,Y 540.586,Z 420.586,A -85,B 0,C 180,E1 26031.368,E2 26031.368} C_VEL
LIN {X 0,Y 539.965,Z 438.228,A -85,B 0,C 180,E1 26030.541,E2 26030.541} C_VEL
LIN {X 0,Y 539.297,Z 454.826,A -85,B 0,C 180,E1 26029.55,E2 26029.55} C_VEL
LIN {X 0,Y 538.578,Z 471.219,A -85,B 0,C 180,E1 26028.34,E2 26028.34} C_VEL
LIN {X 0,Y 537.886,Z 486.426,A -85,B 0,C 180,E1 26026.967,E2 26026.967} C_VEL
LIN {X 0,Y 537.311,Z 499.583,A -85,B 0,C 180,E1 26025.542,E2 26025.542} C_VEL
LIN {X 0,Y 536.79,Z 512.199,A -85,B 0,C 180,E1 26023.902,E2 26023.902} C_VEL
LIN {X 0,Y 536.402,Z 523.969,A -85,B 0,C 180,E1 26022.049,E2 26022.049} C_VEL
LIN {X 0,Y 536.174,Z 533.782,A -85,B 0,C 180,E1 26020.203,E2 26020.203} C_VEL
LIN {X 0,Y 536.032,Z 542.012,A -85,B 0,C 180,E1 26018.257,E2 26018.257} C_VEL
LIN {X 0,Y 535.95,Z 548.29,A -85,B 0,C 180,E1 26016.319,E2 26016.319} C_VEL
LIN {X 0,Y 535.922,Z 552.79,A -85,B 0,C 180,E1 26014.386,E2 26014.386} C_VEL
LIN {X 0,Y 535.912,Z 555.744,A -85,B 0,C 180,E1 26012.352,E2 26012.352} C_VEL
LIN {X 0,Y 535.909,Z 556.93,A -85,B 0,C 180,E1 26010.32,E2 26010.32} C_VEL
LIN {X 0,Y 535.914,Z 556.374,A -85,B 0,C 180,E1 26008.289,E2 26008.289} C_VEL
LIN {X 0,Y 535.911,Z 554.226,A -85,B 0,C 180,E1 26006.362,E2 26006.362} C_VEL
LIN {X 0,Y 535.936,Z 550.454,A -85,B 0,C 180,E1 26004.432,E2 26004.432} C_VEL
LIN {X 0,Y 535.984,Z 544.963,A -85,B 0,C 180,E1 26002.496,E2 26002.496} C_VEL
LIN {X 0,Y 536.097,Z 537.612,A -85,B 0,C 180,E1 26000.553,E2 26000.553} C_VEL
LIN {X 0,Y 536.282,Z 528.749,A -85,B 0,C 180,E1 25998.71,E2 25998.71} C_VEL
LIN {X 0,Y 536.642,Z 516.512,A -85,B 0,C 180,E1 25996.641,E2 25996.641} C_VEL
LIN {X 0,Y 537.097,Z 504.766,A -85,B 0,C 180,E1 25995.003,E2 25995.003} C_VEL
LIN {X 0,Y 537.686,Z 491.024,A -85,B 0,C 180,E1 25993.414,E2 25993.414} C_VEL
LIN {X 0,Y 538.322,Z 476.75,A -85,B 0,C 180,E1 25992.041,E2 25992.041} C_VEL
LIN {X 0,Y 539.004,Z 461.581,A -85,B 0,C 180,E1 25990.832,E2 25990.832} C_VEL
LIN {X 0,Y 539.674,Z 445.627,A -85,B 0,C 180,E1 25989.785,E2 25989.785} C_VEL
LIN {X 0,Y 540.307,Z 428.864,A -85,B 0,C 180,E1 25988.904,E2 25988.904} C_VEL
LIN {X 0,Y 540.859,Z 411.002,A -85,B 0,C 180,E1 25988.182,E2 25988.182} C_VEL
LIN {X 0,Y 541.28,Z 392.628,A -85,B 0,C 180,E1 25987.651,E2 25987.651} C_VEL
LIN {X 0,Y 541.522,Z 372.816,A -85,B 0,C 180,E1 25987.293,E2 25987.293} C_VEL
LIN {X 0,Y 542.489,Z 185.194,A -85,B 0,C 180,E1 25984.708,E2 25984.708} C_VEL
LIN {X 0,Y 540.57,Z 174.378,A -85,B 0,C 180,E1 25984.412,E2 25984.412} C_VEL
LIN {X 0,Y 541.83,Z 134.783,A -85,B 0,C 180,E1 25981.087,E2 25981.087} C_VEL
LIN {X 0,Y 542.2,Z 119.561,A -85,B 0,C 180,E1 25979.772,E2 25979.772} C_VEL
LIN {X 0,Y 536.406,Z 102.671,A -85,B 0,C 180,E1 25977.833,E2 25977.833} C_VEL
LIN {X 0,Y 536.408,Z 102.665,A -85,B 0,C 180,E1 25974.439,E2 25974.439} C_VEL
LIN {X 0,Y 536.46,Z 102.644,A -85,B 0,C 180,E1 25971.176,E2 25971.176} C_VEL
LIN {X 0,Y 536.459,Z 102.666,A -85,B 0,C 180,E1 25967.857,E2 25967.857} C_VEL
LIN {X 0,Y 536.44,Z 102.664,A -85,B 0,C 180,E1 25964.449,E2 25964.449} C_VEL
LIN {X 0,Y 536.453,Z 102.659,A -85,B 0,C 180,E1 25960.987,E2 25960.987} C_VEL
LIN {X 0,Y 536.452,Z 102.659,A -85,B 0,C 180,E1 25957.614,E2 25957.614} C_VEL
LIN {X 0,Y 536.446,Z 102.665,A -85,B 0,C 180,E1 25954.127,E2 25954.127} C_VEL
LIN {X 0,Y 536.468,Z 102.736,A -85,B 0,C 180,E1 25951.429,E2 25951.429} C_VEL
LIN {X 0,Y 541.219,Z 117.905,A -85,B 0,C 180,E1 25949.921,E2 25949.921} C_VEL
LIN {X 0,Y 540.53,Z 158.687,A -85,B 0,C 180,E1 25946.658,E2 25946.658} C_VEL
LIN {X 0,Y 540.275,Z 177.667,A -85,B 0,C 180,E1 25945.165,E2 25945.165} C_VEL
LIN {X 0,Y 541.563,Z 187.163,A -85,B 0,C 180,E1 25944.958,E2 25944.958} C_VEL
LIN {X 0,Y 540.234,Z 386.042,A -85,B 0,C 180,E1 25942.115,E2 25942.115} C_VEL
LIN {X 0,Y 539.966,Z 404.802,A -85,B 0,C 180,E1 25941.655,E2 25941.655} C_VEL
LIN {X 0,Y 539.577,Z 423.671,A -85,B 0,C 180,E1 25940.984,E2 25940.984} C_VEL
LIN {X 0,Y 539.097,Z 441.699,A -85,B 0,C 180,E1 25940.124,E2 25940.124} C_VEL
LIN {X 0,Y 538.572,Z 458.989,A -85,B 0,C 180,E1 25939.072,E2 25939.072} C_VEL
LIN {X 0,Y 538.006,Z 475.757,A -85,B 0,C 180,E1 25937.801,E2 25937.801} C_VEL
LIN {X 0,Y 537.511,Z 489.876,A -85,B 0,C 180,E1 25936.504,E2 25936.504} C_VEL
LIN {X 0,Y 537.037,Z 503.448,A -85,B 0,C 180,E1 25934.999,E2 25934.999} C_VEL
LIN {X 0,Y 536.677,Z 514.154,A -85,B 0,C 180,E1 25933.577,E2 25933.577} C_VEL
LIN {X 0,Y 536.372,Z 525.253,A -85,B 0,C 180,E1 25931.833,E2 25931.833} C_VEL
LIN {X 0,Y 536.166,Z 533.735,A -85,B 0,C 180,E1 25930.205,E2 25930.205} C_VEL
LIN {X 0,Y 536.044,Z 541.197,A -85,B 0,C 180,E1 25928.474,E2 25928.474} C_VEL
LIN {X 0,Y 535.965,Z 547.664,A -85,B 0,C 180,E1 25926.534,E2 25926.534} C_VEL
LIN {X 0,Y 535.922,Z 551.903,A -85,B 0,C 180,E1 25924.816,E2 25924.816} C_VEL
LIN {X 0,Y 535.917,Z 555.181,A -85,B 0,C 180,E1 25922.888,E2 25922.888} C_VEL
LIN {X 0,Y 535.912,Z 556.755,A -85,B 0,C 180,E1 25920.855,E2 25920.855} C_VEL
LIN {X 0,Y 535.911,Z 556.765,A -85,B 0,C 180,E1 25919.038,E2 25919.038} C_VEL
LIN {X 0,Y 535.915,Z 554.966,A -85,B 0,C 180,E1 25916.899,E2 25916.899} C_VEL
LIN {X 0,Y 535.923,Z 552.088,A -85,B 0,C 180,E1 25915.184,E2 25915.184} C_VEL
LIN {X 0,Y 535.963,Z 547.359,A -85,B 0,C 180,E1 25913.251,E2 25913.251} C_VEL
LIN {X 0,Y 536.042,Z 540.782,A -85,B 0,C 180,E1 25911.338,E2 25911.338} C_VEL
LIN {X 0,Y 536.169,Z 533.672,A -85,B 0,C 180,E1 25909.687,E2 25909.687} C_VEL
LIN {X 0,Y 536.401,Z 523.835,A -85,B 0,C 180,E1 25907.841,E2 25907.841} C_VEL
LIN {X 0,Y 536.71,Z 513.294,A -85,B 0,C 180,E1 25906.205,E2 25906.205} C_VEL
LIN {X 0,Y 537.143,Z 500.594,A -85,B 0,C 180,E1 25904.563,E2 25904.563} C_VEL
LIN {X 0,Y 537.609,Z 487.167,A -85,B 0,C 180,E1 25903.134,E2 25903.134} C_VEL
LIN {X 0,Y 538.123,Z 472.15,A -85,B 0,C 180,E1 25901.811,E2 25901.811} C_VEL
LIN {X 0,Y 538.607,Z 456.841,A -85,B 0,C 180,E1 25900.705,E2 25900.705} C_VEL
LIN {X 0,Y 539.084,Z 439.685,A -85,B 0,C 180,E1 25899.706,E2 25899.706} C_VEL
LIN {X 0,Y 539.493,Z 421.974,A -85,B 0,C 180,E1 25898.899,E2 25898.899} C_VEL
LIN {X 0,Y 539.807,Z 403.582,A -85,B 0,C 180,E1 25898.275,E2 25898.275} C_VEL
LIN {X 0,Y 540.029,Z 384.312,A -85,B 0,C 180,E1 25897.834,E2 25897.834} C_VEL
LIN {X 0,Y 541.279,Z 195.503,A -85,B 0,C 180,E1 25895.143,E2 25895.143} C_VEL
LIN {X 0,Y 541.132,Z 184.147,A -85,B 0,C 180,E1 25894.963,E2 25894.963} C_VEL
LIN {X 0,Y 540.36,Z 179.335,A -85,B 0,C 180,E1 25894.842,E2 25894.842} C_VEL
LIN {X 0,Y 540.625,Z 142.63,A -85,B 0,C 180,E1 25892.041,E2 25892.041} C_VEL
LIN {X 0,Y 540.526,Z 116.303,A -85,B 0,C 180,E1 25890.098,E2 25890.098} C_VEL
LIN {X 0,Y 536.444,Z 102.667,A -85,B 0,C 180,E1 25888.885,E2 25888.885} C_VEL
LIN {X 0,Y 536.467,Z 102.664,A -85,B 0,C 180,E1 25885.487,E2 25885.487} C_VEL
LIN {X 0,Y 536.423,Z 102.664,A -85,B 0,C 180,E1 25882.176,E2 25882.176} C_VEL
LIN {X 0,Y 536.409,Z 102.666,A -85,B 0,C 180,E1 25878.854,E2 25878.854} C_VEL
LIN {X 0,Y 536.453,Z 102.666,A -85,B 0,C 180,E1 25875.55,E2 25875.55} C_VEL
LIN {X 0,Y 536.406,Z 102.667,A -85,B 0,C 180,E1 25872.268,E2 25872.268} C_VEL
LIN {X 0,Y 536.391,Z 102.669,A -85,B 0,C 180,E1 25868.917,E2 25868.917} C_VEL
LIN {X 0,Y 536.459,Z 102.672,A -85,B 0,C 180,E1 25865.927,E2 25865.927} C_VEL
LIN {X 0,Y 544.112,Z 122.684,A -85,B 0,C 180,E1 25863.997,E2 25863.997} C_VEL
LIN {X 0,Y 543.202,Z 163.502,A -85,B 0,C 180,E1 25861.317,E2 25861.317} C_VEL
LIN {X 0,Y 544.955,Z 175.575,A -85,B 0,C 180,E1 25861.032,E2 25861.032} C_VEL
LIN {X 0,Y 543.084,Z 414.398,A -85,B 0,C 180,E1 25857.6,E2 25857.6} C_VEL
LIN {X 0,Y 542.753,Z 435.601,A -85,B 0,C 180,E1 25857.197,E2 25857.197} C_VEL
LIN {X 0,Y 542.216,Z 455.754,A -85,B 0,C 180,E1 25856.618,E2 25856.618} C_VEL
LIN {X 0,Y 541.63,Z 474.689,A -85,B 0,C 180,E1 25855.887,E2 25855.887} C_VEL
LIN {X 0,Y 540.94,Z 493.256,A -85,B 0,C 180,E1 25854.984,E2 25854.984} C_VEL
LIN {X 0,Y 540.187,Z 511.982,A -85,B 0,C 180,E1 25853.862,E2 25853.862} C_VEL
LIN {X 0,Y 539.404,Z 529.83,A -85,B 0,C 180,E1 25852.564,E2 25852.564} C_VEL
LIN {X 0,Y 538.641,Z 546.64,A -85,B 0,C 180,E1 25851.108,E2 25851.108} C_VEL
LIN {X 0,Y 537.944,Z 562.449,A -85,B 0,C 180,E1 25849.49,E2 25849.49} C_VEL
LIN {X 0,Y 537.351,Z 576.747,A -85,B 0,C 180,E1 25847.768,E2 25847.768} C_VEL
LIN {X 0,Y 536.86,Z 589.979,A -85,B 0,C 180,E1 25845.89,E2 25845.89} C_VEL
LIN {X 0,Y 536.5,Z 601.108,A -85,B 0,C 180,E1 25844.022,E2 25844.022} C_VEL
LIN {X 0,Y 536.227,Z 611.408,A -85,B 0,C 180,E1 25841.946,E2 25841.946} C_VEL
LIN {X 0,Y 536.062,Z 619.68,A -85,B 0,C 180,E1 25839.881,E2 25839.881} C_VEL
LIN {X 0,Y 535.979,Z 626.2,A -85,B 0,C 180,E1 25837.828,E2 25837.828} C_VEL
LIN {X 0,Y 535.929,Z 631.347,A -85,B 0,C 180,E1 25835.675,E2 25835.675} C_VEL
LIN {X 0,Y 535.908,Z 634.826,A -85,B 0,C 180,E1 25833.531,E2 25833.531} C_VEL
LIN {X 0,Y 535.906,Z 636.707,A -85,B 0,C 180,E1 25831.284,E2 25831.284} C_VEL
LIN {X 0,Y 535.911,Z 636.828,A -85,B 0,C 180,E1 25829.145,E2 25829.145} C_VEL
LIN {X 0,Y 535.913,Z 635.282,A -85,B 0,C 180,E1 25826.899,E2 25826.899} C_VEL
LIN {X 0,Y 535.92,Z 631.967,A -85,B 0,C 180,E1 25824.648,E2 25824.648} C_VEL
LIN {X 0,Y 535.964,Z 627.114,A -85,B 0,C 180,E1 25822.497,E2 25822.497} C_VEL
LIN {X 0,Y 536.054,Z 620.492,A -85,B 0,C 180,E1 25820.337,E2 25820.337} C_VEL
LIN {X 0,Y 536.214,Z 611.879,A -85,B 0,C 180,E1 25818.165,E2 25818.165} C_VEL
LIN {X 0,Y 536.466,Z 602.145,A -85,B 0,C 180,E1 25816.175,E2 25816.175} C_VEL
LIN {X 0,Y 536.838,Z 590.692,A -85,B 0,C 180,E1 25814.222,E2 25814.222} C_VEL
LIN {X 0,Y 537.329,Z 577.357,A -85,B 0,C 180,E1 25812.312,E2 25812.312} C_VEL
LIN {X 0,Y 537.925,Z 562.967,A -85,B 0,C 180,E1 25810.567,E2 25810.567} C_VEL
LIN {X 0,Y 538.597,Z 547.861,A -85,B 0,C 180,E1 25809.006,E2 25809.006} C_VEL
LIN {X 0,Y 539.342,Z 531.285,A -85,B 0,C 180,E1 25807.55,E2 25807.55} C_VEL
LIN {X 0,Y 540.096,Z 513.709,A -85,B 0,C 180,E1 25806.257,E2 25806.257} C_VEL
LIN {X 0,Y 540.841,Z 495.625,A -85,B 0,C 180,E1 25805.149,E2 25805.149} C_VEL
LIN {X 0,Y 541.582,Z 476.001,A -85,B 0,C 180,E1 25804.171,E2 25804.171} C_VEL
LIN {X 0,Y 542.21,Z 456.018,A -85,B 0,C 180,E1 25803.391,E2 25803.391} C_VEL
LIN {X 0,Y 542.75,Z 435.836,A -85,B 0,C 180,E1 25802.808,E2 25802.808} C_VEL
LIN {X 0,Y 543.082,Z 414.621,A -85,B 0,C 180,E1 25802.403,E2 25802.403} C_VEL
LIN {X 0,Y 544.951,Z 175.934,A -85,B 0,C 180,E1 25798.973,E2 25798.973} C_VEL
LIN {X 0,Y 544.153,Z 169.198,A -85,B 0,C 180,E1 25798.821,E2 25798.821} C_VEL
LIN {X 0,Y 543.118,Z 162.609,A -85,B 0,C 180,E1 25798.649,E2 25798.649} C_VEL
LIN {X 0,Y 544.088,Z 122.299,A -85,B 0,C 180,E1 25795.975,E2 25795.975} C_VEL
LIN {X 0,Y 536.466,Z 102.665,A -85,B 0,C 180,E1 25794.05,E2 25794.05} C_VEL
LIN {X 0,Y 536.411,Z 102.663,A -85,B 0,C 180,E1 25790.812,E2 25790.812} C_VEL
LIN {X 0,Y 536.414,Z 102.666,A -85,B 0,C 180,E1 25787.414,E2 25787.414} C_VEL
LIN {X 0,Y 536.466,Z 102.664,A -85,B 0,C 180,E1 25784.148,E2 25784.148} C_VEL
LIN {X 0,Y 536.413,Z 102.662,A -85,B 0,C 180,E1 25780.821,E2 25780.821} C_VEL
LIN {X 0,Y 536.408,Z 102.656,A -85,B 0,C 180,E1 25777.42,E2 25777.42} C_VEL
LIN {X 0,Y 536.462,Z 102.662,A -85,B 0,C 180,E1 25774.125,E2 25774.125} C_VEL
LIN {X 0,Y 536.413,Z 102.664,A -85,B 0,C 180,E1 25770.836,E2 25770.836} C_VEL
LIN {X 0,Y 536.403,Z 102.664,A -85,B 0,C 180,E1 25767.413,E2 25767.413} C_VEL
LIN {X 0,Y 536.453,Z 102.658,A -85,B 0,C 180,E1 25764.09,E2 25764.09} C_VEL
LIN {X 0,Y 536.413,Z 102.664,A -85,B 0,C 180,E1 25760.856,E2 25760.856} C_VEL
LIN {X 0,Y 536.4,Z 102.663,A -85,B 0,C 180,E1 25757.464,E2 25757.464} C_VEL
LIN {X 0,Y 536.461,Z 102.657,A -85,B 0,C 180,E1 25754.242,E2 25754.242} C_VEL
LIN {X 0,Y 536.408,Z 102.663,A -85,B 0,C 180,E1 25750.96,E2 25750.96} C_VEL
LIN {X 0,Y 536.399,Z 102.656,A -85,B 0,C 180,E1 25747.605,E2 25747.605} C_VEL
LIN {X 0,Y 536.456,Z 102.665,A -85,B 0,C 180,E1 25744.344,E2 25744.344} C_VEL
LIN {X 0,Y 536.404,Z 102.657,A -85,B 0,C 180,E1 25741.068,E2 25741.068} C_VEL
LIN {X 0,Y 536.396,Z 102.665,A -85,B 0,C 180,E1 25737.649,E2 25737.649} C_VEL
LIN {X 0,Y 536.448,Z 102.656,A -85,B 0,C 180,E1 25734.331,E2 25734.331} C_VEL
LIN {X 0,Y 536.405,Z 102.665,A -85,B 0,C 180,E1 25731.1,E2 25731.1} C_VEL
LIN {X 0,Y 536.393,Z 102.66,A -85,B 0,C 180,E1 25727.731,E2 25727.731} C_VEL
LIN {X 0,Y 536.452,Z 102.663,A -85,B 0,C 180,E1 25724.431,E2 25724.431} C_VEL
LIN {X 0,Y 536.401,Z 102.66,A -85,B 0,C 180,E1 25721.187,E2 25721.187} C_VEL
LIN {X 0,Y 536.39,Z 102.661,A -85,B 0,C 180,E1 25717.765,E2 25717.765} C_VEL
LIN {X 0,Y 536.447,Z 102.666,A -85,B 0,C 180,E1 25714.497,E2 25714.497} C_VEL
LIN {X 0,Y 536.397,Z 102.657,A -85,B 0,C 180,E1 25711.254,E2 25711.254} C_VEL
LIN {X 0,Y 536.391,Z 102.662,A -85,B 0,C 180,E1 25707.909,E2 25707.909} C_VEL
LIN {X 0,Y 536.39,Z 102.665,A -85,B 0,C 180,E1 25705.417,E2 25705.417} C_VEL
LIN {X 0,Y 535.421,Z 102.793,A -85,B 0,C 180,E1 25704.593,E2 25704.593} C_VEL
LIN {X 0,Y 528.978,Z 103.591,A -85,B 0,C 180,E1 25702.282,E2 25702.282} C_VEL
LIN {X 0,Y 528.446,Z 103.654,A -85,B 0,C 180,E1 25701.679,E2 25701.679} C_VEL
LIN {X 0,Y 528.477,Z 103.656,A -85,B 0,C 180,E1 25698.358,E2 25698.358} C_VEL
LIN {X 0,Y 528.484,Z 103.651,A -85,B 0,C 180,E1 25695.037,E2 25695.037} C_VEL
LIN {X 0,Y 528.445,Z 103.657,A -85,B 0,C 180,E1 25691.759,E2 25691.759} C_VEL
LIN {X 0,Y 528.478,Z 103.654,A -85,B 0,C 180,E1 25688.438,E2 25688.438} C_VEL
LIN {X 0,Y 528.478,Z 103.654,A -85,B 0,C 180,E1 25685.182,E2 25685.182} C_VEL
LIN {X 0,Y 528.504,Z 103.792,A -85,B 0,C 180,E1 25682.53,E2 25682.53} C_VEL
LIN {X 0,Y 535.075,Z 123.13,A -85,B 0,C 180,E1 25680.299,E2 25680.299} C_VEL
LIN {X 0,Y 533.597,Z 163.389,A -85,B 0,C 180,E1 25676.845,E2 25676.845} C_VEL
LIN {X 0,Y 533.314,Z 175.187,A -85,B 0,C 180,E1 25675.879,E2 25675.879} C_VEL
LIN {X 0,Y 535.52,Z 188.028,A -85,B 0,C 180,E1 25675.566,E2 25675.566} C_VEL
LIN {X 0,Y 534.324,Z 384.54,A -85,B 0,C 180,E1 25672.829,E2 25672.829} C_VEL
LIN {X 0,Y 533.95,Z 403.317,A -85,B 0,C 180,E1 25672.377,E2 25672.377} C_VEL
LIN {X 0,Y 533.403,Z 421.604,A -85,B 0,C 180,E1 25671.728,E2 25671.728} C_VEL
LIN {X 0,Y 532.716,Z 439.149,A -85,B 0,C 180,E1 25670.891,E2 25670.891} C_VEL
LIN {X 0,Y 531.97,Z 455.682,A -85,B 0,C 180,E1 25669.888,E2 25669.888} C_VEL
LIN {X 0,Y 531.148,Z 471.973,A -85,B 0,C 180,E1 25668.663,E2 25668.663} C_VEL
LIN {X 0,Y 530.349,Z 487.097,A -85,B 0,C 180,E1 25667.273,E2 25667.273} C_VEL
LIN {X 0,Y 529.652,Z 500.649,A -85,B 0,C 180,E1 25665.773,E2 25665.773} C_VEL
LIN {X 0,Y 529.049,Z 513.174,A -85,B 0,C 180,E1 25664.11,E2 25664.11} C_VEL
LIN {X 0,Y 528.597,Z 524.193,A -85,B 0,C 180,E1 25662.341,E2 25662.341} C_VEL
LIN {X 0,Y 528.268,Z 533.737,A -85,B 0,C 180,E1 25660.468,E2 25660.468} C_VEL
LIN {X 0,Y 528.063,Z 541.77,A -85,B 0,C 180,E1 25658.492,E2 25658.492} C_VEL
LIN {X 0,Y 527.955,Z 548.595,A -85,B 0,C 180,E1 25656.305,E2 25656.305} C_VEL
LIN {X 0,Y 527.923,Z 552.997,A -85,B 0,C 180,E1 25654.344,E2 25654.344} C_VEL
LIN {X 0,Y 527.911,Z 555.744,A -85,B 0,C 180,E1 25652.387,E2 25652.387} C_VEL
LIN {X 0,Y 527.909,Z 556.929,A -85,B 0,C 180,E1 25650.325,E2 25650.325} C_VEL
LIN {X 0,Y 527.914,Z 556.373,A -85,B 0,C 180,E1 25648.263,E2 25648.263} C_VEL
LIN {X 0,Y 527.914,Z 554.224,A -85,B 0,C 180,E1 25646.307,E2 25646.307} C_VEL
LIN {X 0,Y 527.94,Z 550.452,A -85,B 0,C 180,E1 25644.348,E2 25644.348} C_VEL
LIN {X 0,Y 528.017,Z 544.32,A -85,B 0,C 180,E1 25642.163,E2 25642.163} C_VEL
LIN {X 0,Y 528.171,Z 537.026,A -85,B 0,C 180,E1 25640.19,E2 25640.19} C_VEL
LIN {X 0,Y 528.445,Z 528.277,A -85,B 0,C 180,E1 25638.319,E2 25638.319} C_VEL
LIN {X 0,Y 528.878,Z 517.456,A -85,B 0,C 180,E1 25636.442,E2 25636.442} C_VEL
LIN {X 0,Y 529.408,Z 505.804,A -85,B 0,C 180,E1 25634.78,E2 25634.78} C_VEL
LIN {X 0,Y 530.09,Z 492.198,A -85,B 0,C 180,E1 25633.169,E2 25633.169} C_VEL
LIN {X 0,Y 530.854,Z 477.466,A -85,B 0,C 180,E1 25631.723,E2 25631.723} C_VEL
LIN {X 0,Y 531.636,Z 462.388,A -85,B 0,C 180,E1 25630.498,E2 25630.498} C_VEL
LIN {X 0,Y 532.393,Z 446.498,A -85,B 0,C 180,E1 25629.439,E2 25629.439} C_VEL
LIN {X 0,Y 533.12,Z 429.12,A -85,B 0,C 180,E1 25628.516,E2 25628.516} C_VEL
LIN {X 0,Y 533.719,Z 411.326,A -85,B 0,C 180,E1 25627.792,E2 25627.792} C_VEL
LIN {X 0,Y 534.174,Z 393.04,A -85,B 0,C 180,E1 25627.261,E2 25627.261} C_VEL
LIN {X 0,Y 534.427,Z 373.341,A -85,B 0,C 180,E1 25626.903,E2 25626.903} C_VEL
LIN {X 0,Y 535.428,Z 186.342,A -85,B 0,C 180,E1 25624.317,E2 25624.317} C_VEL
LIN {X 0,Y 533.239,Z 174.532,A -85,B 0,C 180,E1 25624.004,E2 25624.004} C_VEL
LIN {X 0,Y 534.672,Z 134.809,A -85,B 0,C 180,E1 25620.627,E2 25620.627} C_VEL
LIN {X 0,Y 535.042,Z 122.74,A -85,B 0,C 180,E1 25619.573,E2 25619.573} C_VEL
LIN {X 0,Y 528.517,Z 103.656,A -85,B 0,C 180,E1 25617.337,E2 25617.337} C_VEL
LIN {X 0,Y 528.481,Z 103.655,A -85,B 0,C 180,E1 25613.956,E2 25613.956} C_VEL
LIN {X 0,Y 528.482,Z 103.636,A -85,B 0,C 180,E1 25610.526,E2 25610.526} C_VEL
LIN {X 0,Y 528.522,Z 103.646,A -85,B 0,C 180,E1 25607.222,E2 25607.222} C_VEL
LIN {X 0,Y 528.523,Z 103.646,A -85,B 0,C 180,E1 25603.724,E2 25603.724} C_VEL
LIN {X 0,Y 528.521,Z 103.652,A -85,B 0,C 180,E1 25600.316,E2 25600.316} C_VEL
LIN {X 0,Y 528.517,Z 103.65,A -85,B 0,C 180,E1 25596.846,E2 25596.846} C_VEL
LIN {X 0,Y 528.52,Z 103.65,A -85,B 0,C 180,E1 25593.403,E2 25593.403} C_VEL
LIN {X 0,Y 528.509,Z 103.73,A -85,B 0,C 180,E1 25591.833,E2 25591.833} C_VEL
LIN {X 0,Y 533.866,Z 121.129,A -85,B 0,C 180,E1 25590.087,E2 25590.087} C_VEL
LIN {X 0,Y 533.076,Z 161.71,A -85,B 0,C 180,E1 25586.814,E2 25586.814} C_VEL
LIN {X 0,Y 532.891,Z 178.224,A -85,B 0,C 180,E1 25585.519,E2 25585.519} C_VEL
LIN {X 0,Y 534.264,Z 188.25,A -85,B 0,C 180,E1 25585.296,E2 25585.296} C_VEL
LIN {X 0,Y 532.698,Z 386.744,A -85,B 0,C 180,E1 25582.394,E2 25582.394} C_VEL
LIN {X 0,Y 532.403,Z 405.668,A -85,B 0,C 180,E1 25581.92,E2 25581.92} C_VEL
LIN {X 0,Y 531.979,Z 424.484,A -85,B 0,C 180,E1 25581.237,E2 25581.237} C_VEL
LIN {X 0,Y 531.457,Z 442.38,A -85,B 0,C 180,E1 25580.368,E2 25580.368} C_VEL
LIN {X 0,Y 530.907,Z 459.036,A -85,B 0,C 180,E1 25579.345,E2 25579.345} C_VEL
LIN {X 0,Y 530.33,Z 474.789,A -85,B 0,C 180,E1 25578.154,E2 25578.154} C_VEL
LIN {X 0,Y 529.755,Z 489.691,A -85,B 0,C 180,E1 25576.785,E2 25576.785} C_VEL
LIN {X 0,Y 529.224,Z 503.7,A -85,B 0,C 180,E1 25575.225,E2 25575.225} C_VEL
LIN {X 0,Y 528.79,Z 515.646,A -85,B 0,C 180,E1 25573.615,E2 25573.615} C_VEL
LIN {X 0,Y 528.431,Z 526.785,A -85,B 0,C 180,E1 25571.792,E2 25571.792} C_VEL
LIN {X 0,Y 528.199,Z 534.966,A -85,B 0,C 180,E1 25570.14,E2 25570.14} C_VEL
LIN {X 0,Y 528.043,Z 542.522,A -85,B 0,C 180,E1 25568.274,E2 25568.274} C_VEL
LIN {X 0,Y 527.957,Z 548.54,A -85,B 0,C 180,E1 25566.306,E2 25566.306} C_VEL
LIN {X 0,Y 527.923,Z 552.804,A -85,B 0,C 180,E1 25564.454,E2 25564.454} C_VEL
LIN {X 0,Y 527.915,Z 555.713,A -85,B 0,C 180,E1 25562.388,E2 25562.388} C_VEL
LIN {X 0,Y 527.918,Z 556.819,A -85,B 0,C 180,E1 25560.651,E2 25560.651} C_VEL
LIN {X 0,Y 527.911,Z 556.675,A -85,B 0,C 180,E1 25558.698,E2 25558.698} C_VEL
LIN {X 0,Y 527.919,Z 554.807,A -85,B 0,C 180,E1 25556.743,E2 25556.743} C_VEL
LIN {X 0,Y 527.921,Z 551.862,A -85,B 0,C 180,E1 25555.002,E2 25555.002} C_VEL
LIN {X 0,Y 527.978,Z 547.038,A -85,B 0,C 180,E1 25553.039,E2 25553.039} C_VEL
LIN {X 0,Y 528.077,Z 540.397,A -85,B 0,C 180,E1 25551.068,E2 25551.068} C_VEL
LIN {X 0,Y 528.282,Z 532.46,A -85,B 0,C 180,E1 25549.201,E2 25549.201} C_VEL
LIN {X 0,Y 528.563,Z 522.981,A -85,B 0,C 180,E1 25547.436,E2 25547.436} C_VEL
LIN {X 0,Y 528.938,Z 512.194,A -85,B 0,C 180,E1 25545.775,E2 25545.775} C_VEL
LIN {X 0,Y 529.406,Z 499.533,A -85,B 0,C 180,E1 25544.175,E2 25544.175} C_VEL
LIN {X 0,Y 529.907,Z 486.126,A -85,B 0,C 180,E1 25542.769,E2 25542.769} C_VEL
LIN {X 0,Y 530.45,Z 471.093,A -85,B 0,C 180,E1 25541.464,E2 25541.464} C_VEL
LIN {X 0,Y 530.984,Z 454.787,A -85,B 0,C 180,E1 25540.309,E2 25540.309} C_VEL
LIN {X 0,Y 531.476,Z 437.84,A -85,B 0,C 180,E1 25539.345,E2 25539.345} C_VEL
LIN {X 0,Y 531.897,Z 419.844,A -85,B 0,C 180,E1 25538.549,E2 25538.549} C_VEL
LIN {X 0,Y 532.219,Z 401.326,A -85,B 0,C 180,E1 25537.946,E2 25537.946} C_VEL
LIN {X 0,Y 532.431,Z 382.398,A -85,B 0,C 180,E1 25537.537,E2 25537.537} C_VEL
LIN {X 0,Y 533.633,Z 220.259,A -85,B 0,C 180,E1 25535.188,E2 25535.188} C_VEL
LIN {X 0,Y 533.808,Z 185.428,A -85,B 0,C 180,E1 25534.641,E2 25534.641} C_VEL
LIN {X 0,Y 533.011,Z 180.39,A -85,B 0,C 180,E1 25534.511,E2 25534.511} C_VEL
LIN {X 0,Y 533.271,Z 145.769,A -85,B 0,C 180,E1 25531.865,E2 25531.865} C_VEL
LIN {X 0,Y 533.012,Z 118.253,A -85,B 0,C 180,E1 25529.819,E2 25529.819} C_VEL
LIN {X 0,Y 528.487,Z 103.657,A -85,B 0,C 180,E1 25528.49,E2 25528.49} C_VEL
LIN {X 0,Y 528.51,Z 103.655,A -85,B 0,C 180,E1 25525.157,E2 25525.157} C_VEL
LIN {X 0,Y 528.516,Z 103.653,A -85,B 0,C 180,E1 25521.784,E2 25521.784} C_VEL
LIN {X 0,Y 528.465,Z 103.655,A -85,B 0,C 180,E1 25518.525,E2 25518.525} C_VEL
LIN {X 0,Y 528.472,Z 103.657,A -85,B 0,C 180,E1 25515.113,E2 25515.113} C_VEL
LIN {X 0,Y 528.511,Z 103.654,A -85,B 0,C 180,E1 25511.754,E2 25511.754} C_VEL
LIN {X 0,Y 528.463,Z 103.658,A -85,B 0,C 180,E1 25508.437,E2 25508.437} C_VEL
LIN {X 0,Y 528.501,Z 103.865,A -85,B 0,C 180,E1 25506.419,E2 25506.419} C_VEL
LIN {X 0,Y 536.958,Z 125.355,A -85,B 0,C 180,E1 25504.283,E2 25504.283} C_VEL
LIN {X 0,Y 535.995,Z 163.654,A -85,B 0,C 180,E1 25501.731,E2 25501.731} C_VEL
LIN {X 0,Y 537.906,Z 176.86,A -85,B 0,C 180,E1 25501.419,E2 25501.419} C_VEL
LIN {X 0,Y 536.299,Z 378.517,A -85,B 0,C 180,E1 25498.514,E2 25498.514} C_VEL
LIN {X 0,Y 535.821,Z 426.675,A -85,B 0,C 180,E1 25497.786,E2 25497.786} C_VEL
LIN {X 0,Y 535.308,Z 447.702,A -85,B 0,C 180,E1 25497.265,E2 25497.265} C_VEL
LIN {X 0,Y 534.654,Z 467.173,A -85,B 0,C 180,E1 25496.582,E2 25496.582} C_VEL
LIN {X 0,Y 533.898,Z 486.607,A -85,B 0,C 180,E1 25495.699,E2 25495.699} C_VEL
LIN {X 0,Y 533.019,Z 505.817,A -85,B 0,C 180,E1 25494.61,E2 25494.61} C_VEL
LIN {X 0,Y 532.156,Z 523.965,A -85,B 0,C 180,E1 25493.357,E2 25493.357} C_VEL
LIN {X 0,Y 531.342,Z 540.56,A -85,B 0,C 180,E1 25491.992,E2 25491.992} C_VEL
LIN {X 0,Y 530.499,Z 557.434,A -85,B 0,C 180,E1 25490.342,E2 25490.342} C_VEL
